// TIA Portal V15.1 program export: 6 tag tables, 0 data types, 10 data blocks, 37 code blocks (in call order from the OBs), 86 instance data blocks

VAR_GLOBAL   // PLC tag table "Analog"
   AI_AG AT %IW68 : Int;
   AI_FD AT %IW70 : Int;
   AI_AP AT %IW72 : Int;
   AI_SB AT %IW74 : Int;
   AI_TEMP_TL AT %IW76 : Int;
   AI_TEMP_AG AT %IW78 : Int;
   AI_TEMP_TS AT %IW80 : Int;
   AI_TEMP_AP AT %IW82 : Int;
   BT_SPAN_Riasing AT %M2.0 : Bool;
   BT_ZERO_Raising AT %M2.1 : Bool;
   MANUAL_Raissing AT %M2.2 : Bool;
   AI_IND_AGG1 AT %IW100 : Int;
   AI_IND_AGG2 AT %IW102 : Int;
   AI_IND_AGG3 AT %IW104 : Int;
   AI_IND_AGG4 AT %IW106 : Int;
   AI_IND_AGG5 AT %IW108 : Int;
END_VAR

VAR_GLOBAL   // PLC tag table "Default tag table"
END_VAR

VAR_GLOBAL   // PLC tag table "Default tag table_1"
   System_Byte AT %MB1 : Byte;
   FirstScan AT %M1.0 : Bool;
   DiagStatusUpdate AT %M1.1 : Bool;
   AlwaysTRUE AT %M1.2 : Bool;
   AlwaysFALSE AT %M1.3 : Bool;
   Clock_Byte AT %MB0 : Byte;
   Clock_10Hz AT %M0.0 : Bool;
   Clock_5Hz AT %M0.1 : Bool;
   "Clock_2.5Hz" AT %M0.2 : Bool;
   Clock_2Hz AT %M0.3 : Bool;
   "Clock_1.25Hz" AT %M0.4 : Bool;
   Clock_1Hz AT %M0.5 : Bool;
   "Clock_0.625Hz" AT %M0.6 : Bool;
   "Clock_0.5Hz" AT %M0.7 : Bool;
   "NAP LIEU" AT %M200.0 : Bool;
   "RUA NOI" AT %M200.1 : Bool;
   TH_NAP_WAG AT %M300.0 : Bool;
   TH_NAP_WAP AT %M300.2 : Bool;
   TH_NAP_WFD AT %M300.1 : Bool;
   TH_NAP_WSB AT %M300.3 : Bool;
   "LUU_CAN TAY" AT %M200.2 : Bool;
   "LUU TAY CEM1" AT %M200.3 : Bool;
   "LUU TAY CEM2" AT %M200.4 : Bool;
   "LUU TAY WAT1" AT %M200.5 : Bool;
   "LUU TAY ADD1" AT %M200.6 : Bool;
   XA_HET_AGG AT %M200.7 : Bool;
   "LUU TAY WAG1" AT %M210.0 : Bool;
   "LUU TAY WAG2" AT %M210.1 : Bool;
   "LUU TAY WAG3" AT %M210.2 : Bool;
   "LUU TAY WAG4" AT %M210.3 : Bool;
   "LUU TAY WAG5" AT %M210.4 : Bool;
END_VAR
VAR_GLOBAL CONSTANT   // user constants
   "Local(1)" : Hw_SubModule := 50;
   "Local~PROFINET_interface_1(1)" : Hw_Interface := 64;
   "Local~PROFINET_interface_1~Port_1(1)" : Hw_Interface := 65;
   "Local~HSC_1(1)" : Hw_Hsc := 257;
   "Local~HSC_2(1)" : Hw_Hsc := 258;
   "Local~HSC_3(1)" : Hw_Hsc := 259;
   "Local~HSC_4(1)" : Hw_Hsc := 260;
   "Local~HSC_5(1)" : Hw_Hsc := 261;
   "Local~HSC_6(1)" : Hw_Hsc := 262;
   "Local~AI_2_1(1)" : Hw_SubModule := 263;
   "Local~DI_14_DQ_10_1(1)" : Hw_SubModule := 264;
   "Local~Pulse_1(1)" : Hw_Pwm := 265;
   "Local~Pulse_2(1)" : Hw_Pwm := 266;
   "OB_Main_P1(1)" : OB_PCYCLE := 1;
   "Local~Pulse_3(1)" : Hw_Pwm := 267;
   "Local~Pulse_4(1)" : Hw_Pwm := 268;
   "None(1)" : Pip := 65535;
   "Automatic update(1)" : Pip := 0;
   "PIP 1(1)" : Pip := 1;
   "PIP 2(1)" : Pip := 2;
   "PIP 3(1)" : Pip := 3;
   "PIP 4(1)" : Pip := 4;
   "PIP OB Servo(1)" : Pip := 32768;
   "Local~DQ_8xRelay_1(1)" : Hw_SubModule := 273;
   "Local~AI_4x13BIT_1(1)" : Hw_SubModule := 271;
   "Local~AI_4xTC_1(1)" : Hw_SubModule := 272;
   "Local~DI_8_DQ_8x24VDC_1" : Hw_SubModule := 274;
   "Local~DQ_16xRelay_1(1)" : Hw_SubModule := 269;
   "Local~AI_4x13BIT_2(1)" : Hw_SubModule := 270;
END_VAR

VAR_GLOBAL   // PLC tag table "In_Put"
   "I_TH. NOI TRON" AT %I0.0 : Bool;   // Input_Tín hiệu nồi trộn
   "I_TH. BTX" AT %I0.1 : Bool;   // Input_Tín hiệu băng tải xiên
   "I_TH. BTN" AT %I0.2 : Bool;   // Input_Tín hiệu băng tải ngang
   "I_TH. TANG SAY" AT %I0.3 : Bool;   // Input_Tín hiệu tang sấy cốt liệu
   "I_TH. GAU COT LIEU" AT %I0.4 : Bool;   // Input_Tín hiệu gàu tải cốt liệu nóng
   "I_TH. GAU F/D" AT %I0.5 : Bool;   // Input_Tín hiệu gàu tải phụ gia bột
   "I_TH. SANG RUNG" AT %I0.6 : Bool;   // Input_Tín hiệu sàng rung cốt liệu nóng
   "I_TH. CUA DONG" AT %I0.7 : Bool;   // Input_Tín hiệu cửa nồi trộn đóng
   "I_TH. CUA MO" AT %I1.0 : Bool;   // Input_Tín hiệu cửa nồi trộn mở
   "I_TH. MNK" AT %I1.1 : Bool;   // Input_Tín hiệu máy nén khí chạy
   "I_TH. TRAN AG1" AT %I1.2 : Bool;   // Input_Tín hiệu báo tràn silo AG1
   "I_TH. TRAN AG2" AT %I1.3 : Bool;   // Input_Tín hiệu báo tràn silo AG2
   "I_TH. TRAN AG3" AT %I1.4 : Bool;   // Input_Tín hiệu báo tràn silo AG3
   "I_TH. TRAN AG4" AT %I1.5 : Bool;   // Input_Tín hiệu báo tràn silo AG4
   "I_TH. TRAN AG5" AT %I2.0 : Bool;   // Input_Tín hiệu báo tràn silo AG5
   "I_TH. TRAN FD1" AT %I2.1 : Bool;   // Input_Tín hiệu báo tràn silo F/D
   "I_TH. TRAN SB1" AT %I2.2 : Bool;   // Input_Tín hiệu báo tràn silo SBS
   "I_TH. SILO FD HIGHT" AT %I2.3 : Bool;   // Input_Tín hiệu báo mức cao silo chứa F/D
   "I_TH. SILO FD LOW" AT %I2.4 : Bool;   // Input_Tín hiệu báo mức thấp silo chứa F/D
   "TH. NOI TRON" AT %M400.0 : Bool;   // Tín hiệu nồi trộn
   "TH. BTX" AT %M400.1 : Bool;   // Tín hiệu băng tải xiên
   "TH. BTN" AT %M400.2 : Bool;   // Tín hiệu băng tải ngang
   "TH. TANG SAY" AT %M400.3 : Bool;   // Tín hiệu tang sấy cốt liệu
   "TH. GAU COT LIEU" AT %M400.4 : Bool;   // Tín hiệu gàu tải cốt liệu nóng
   "TH. GAU F/D" AT %M400.5 : Bool;   // Tín hiệu gàu tải phụ gia bột
   "TH. SANG RUNG" AT %M400.6 : Bool;   // Tín hiệu sàng rung cốt liệu nóng
   "TH. CUA DONG" AT %M400.7 : Bool;   // Tín hiệu cửa nồi trộn đóng
   "TH. CUA MO" AT %M401.0 : Bool;   // Tín hiệu cửa nồi trộn mở
   "TH. MNK" AT %M401.1 : Bool;   // Tín hiệu máy nén khí chạy
   "TH. TRAN AG1" AT %M401.2 : Bool;   // Tín hiệu báo tràn silo AG1
   "TH. TRAN AG2" AT %M401.3 : Bool;   // Tín hiệu báo tràn silo AG2
   "TH. TRAN AG3" AT %M401.4 : Bool;   // Tín hiệu báo tràn silo AG3
   "TH. TRAN AG4" AT %M401.5 : Bool;   // Tín hiệu báo tràn silo AG4
   "TH. TRAN AG5" AT %M401.6 : Bool;   // Tín hiệu báo tràn silo AG5
   "TH. TRAN FD1" AT %M401.7 : Bool;   // Tín hiệu báo tràn silo F/D
   "TH. TRAN SB1" AT %M402.0 : Bool;   // Tín hiệu báo tràn silo SBS
   "TH. SILO FD HIGHT" AT %M402.1 : Bool;   // Tín hiệu báo mức cao silo chứa F/D
   "TH. SILO FD LOW" AT %M402.2 : Bool;   // Tín hiệu báo mức thấp silo chứa F/D
   "TH_CNM SIM" AT %M402.3 : Bool;
   "TH_CND SIM" AT %M402.4 : Bool;
END_VAR

VAR_GLOBAL   // PLC tag table "Out_Put"
   "Q_CAN AP1" AT %Q4.0 : Bool;   // Output_Nồi trộn
   "Q_GAU COT LIEU" AT %Q0.5 : Bool;   // Output_Băng tải xiên
   Q_BTX AT %Q0.1 : Bool;   // Output_Băng tải ngang
   Q_BTN AT %Q0.2 : Bool;   // Output_Tang sấy cốt liệu
   "Q_TANG SAY" AT %Q0.3 : Bool;   // Output_Bơm dầu DO
   "Q_XA W_AG1" AT %Q4.2 : Bool;   // Output_Gàu tải cốt liệu nóng
   "Q_XA W_SB1" AT %Q4.5 : Bool;   // Output_Sàn rung cốt liệu
   "Q_BOM NUOC" AT %Q2.1 : Bool;   // Output_Gàu tải phụ F/D
   "Q_MO CUA" AT %Q2.2 : Bool;   // Output_Vít tải F/D
   "Q_XA CL5" AT %Q3.1 : Bool;   // Output_Bơm nạp hạt nhựa SBS
   "Q_DONG CUA" AT %Q2.3 : Bool;   // Output_Quạt gió lọc bụi
   Q_MNK AT %Q2.4 : Bool;   // Output_Bơm nước lọc bụi
   "Q_BOM SBS" AT %Q1.1 : Bool;   // Output_Van mở cửa nồi trộn
   "Q_CAN AG1" AT %Q3.2 : Bool;   // Output_Van đóng cửa nồi trộn
   "Q_VIT TAI FD" AT %Q1.0 : Bool;   // Output_Máy nén khí
   "Q_XA CL1" AT %Q2.5 : Bool;   // Output_Băng tải xả cốt liệu 1
   "Q_XA CL2" AT %Q2.6 : Bool;   // Output_Băng tải xả cốt liệu 2
   "Q_CAN AG2" AT %Q3.3 : Bool;   // Output_Băng tải xả cốt liệu 3
   "Q_XA CL3" AT %Q2.7 : Bool;   // Output_Băng tải xả cốt liệu 4
   "Q_XA CL4" AT %Q3.0 : Bool;   // Output_Băng tải xả cốt liệu 5
   "Q_CAN AG3" AT %Q3.4 : Bool;   // Output_Van cân AG1
   "Q_CAN AG4" AT %Q3.5 : Bool;   // Output_Van cân AG2
   "Q_CAN AG5" AT %Q3.6 : Bool;   // Output_Van cân AG3
   "Q_SAN RUNG" AT %Q0.6 : Bool;   // Output_Van cân AG4
   "Q_CAN FD1" AT %Q3.7 : Bool;   // Output_Van cân AG5
   "Q_CAN SB1" AT %Q4.1 : Bool;   // Output_Van cân F/D
   "Q_NOI TRON" AT %Q0.0 : Bool;   // Output_Bơm nhựa
   "Q_XA W_AP1" AT %Q4.4 : Bool;   // Output_Van cân hạt nhựa SBS
   "Q_XA W_FD1" AT %Q4.3 : Bool;   // Output_Van xả cân AG1
   "Q_BOM TUOI NHUA" AT %Q4.6 : Bool;   // Output_Van xả cân FD1
   "Q_DAU DOT" AT %Q4.7 : Bool;   // Output_Van xả cân AP1
   "Q_VAN XA SBS" AT %Q5.0 : Bool;   // Output_Van xả cân SB1
   "Q_Rung CL1" AT %Q5.1 : Bool;   // Output_Bổ ssung 1
   "Q_Rung CL2" AT %Q5.2 : Bool;   // Output_Bổ ssung 2
   "Q_Rung CL3" AT %Q5.3 : Bool;   // Output_Bổ ssung 3
   "Q_NOTE 7" AT %Q5.4 : Bool;   // Output_Bổ ssung 4
   "Q_QUAT GIO" AT %Q2.0 : Bool;   // Output_Bổ ssung 5
   "Q_GAU FD" AT %Q0.7 : Bool;   // Output_Bổ ssung 6
   "Q_BOM DAU" AT %Q0.4 : Bool;   // Output_Bổ ssung 7
   "NOI TRON" AT %M500.0 : Bool;   // Nồi trộn
   BTX AT %M500.1 : Bool;   // Băng tải xiên
   BTN AT %M500.2 : Bool;   // Băng tải ngang
   "TANG SAY" AT %M500.3 : Bool;   // Tang sấy cốt liệu
   "BOM DAU" AT %M500.4 : Bool;   // Bơm dầu DO
   "GAU COT LIEU" AT %M500.5 : Bool;   // Gàu tải cốt liệu nóng
   "SAN RUNG" AT %M500.6 : Bool;   // Sàn rung cốt liệu
   "GAU FD" AT %M500.7 : Bool;   // Gàu tải phụ F/D
   "VIT TAI FD" AT %M501.0 : Bool;   // Vít tải F/D
   "BOM SBS" AT %M501.1 : Bool;   // Bơm nạp hạt nhựa SBS
   "QUAT GIO" AT %M501.2 : Bool;   // Quạt gió lọc bụi
   "BOM NUOC" AT %M501.3 : Bool;   // Bơm nước lọc bụi
   "MO CUA" AT %M501.4 : Bool;   // Van mở cửa nồi trộn
   "DONG CUA" AT %M501.5 : Bool;   // Van đóng cửa nồi trộn
   MNK AT %M501.6 : Bool;   // Máy nén khí
   "XA CL1" AT %M501.7 : Bool;   // Băng tải xả cốt liệu 1
   "XA CL2" AT %M502.0 : Bool;   // Băng tải xả cốt liệu 2
   "XA CL3" AT %M502.1 : Bool;   // Băng tải xả cốt liệu 3
   "XA CL4" AT %M502.2 : Bool;   // Băng tải xả cốt liệu 4
   "XA CL5" AT %M502.3 : Bool;   // Băng tải xả cốt liệu 5
   "CAN AG1" AT %M502.4 : Bool;   // Van cân AG1
   "CAN AG2" AT %M502.5 : Bool;   // Van cân AG2
   "CAN AG3" AT %M502.6 : Bool;   // Van cân AG3
   "CAN AG4" AT %M502.7 : Bool;   // Van cân AG4
   "CAN AG5" AT %M503.0 : Bool;   // Van cân AG5
   "CAN FD1" AT %M503.1 : Bool;   // Van cân F/D
   "CAN AP1" AT %M503.2 : Bool;   // Bơm nhựa
   "CAN SB1" AT %M503.3 : Bool;   // Van cân hạt nhựa SBS
   "XA W_AG1" AT %M503.4 : Bool;   // Van xả cân AG1
   "XA W_FD1" AT %M503.5 : Bool;   // Van xả cân FD1
   "XA W_AP1" AT %M503.6 : Bool;   // Van xả cân AP1
   "XA W_SB1" AT %M503.7 : Bool;   // Van xả cân SB1
   "BOM TUOI NHUA" AT %M504.0 : Bool;   // Bổ ssung 1
   "DAU DOT" AT %M504.1 : Bool;   // Bổ ssung 2
   "VAN XA SBS" AT %M504.2 : Bool;   // Bổ ssung 3
   "RUNG CL1" AT %M504.3 : Bool;   // Bổ ssung 4
   "RUNG CL2" AT %M504.4 : Bool;   // Bổ ssung 5
   "RUNG CL3" AT %M504.5 : Bool;   // Bổ ssung 6
   "NOTE 7" AT %M504.6 : Bool;   // Bổ ssung 7
   "Q_XA W_IND AGG1" AT %Q6.0 : Bool;   // Mode=độc lập, Van xả cấn AGG1
   "Q_XA W_IND AGG2" AT %Q6.1 : Bool;   // Mode=độc lập, Van xả cấn AGG2
   "Q_XA W_IND AGG3" AT %Q6.2 : Bool;   // Mode=độc lập, Van xả cấn AGG3
   "Q_XA W_IND AGG4" AT %Q6.3 : Bool;   // Mode=độc lập, Van xả cấn AGG4
   "Q_XA W_IND AGG5" AT %Q6.4 : Bool;   // Mode=độc lập, Van xả cấn AGG5
END_VAR

VAR_GLOBAL   // PLC tag table "XUNG_TEMP"
   P_AGG1_EM AT %M100.0 : Bool;
   P_AGG2_EM AT %M100.1 : Bool;
   P_AGG3_EM AT %M100.2 : Bool;
   P_AGG4_EM AT %M100.3 : Bool;
   P_AGG5_EM AT %M100.4 : Bool;
   P_AGG6_EM AT %M100.5 : Bool;
   P_CE1_EM AT %M100.6 : Bool;
   P_CE2_EM AT %M100.7 : Bool;
   P_CE3_EM AT %M101.0 : Bool;
   P_CE4_EM AT %M101.1 : Bool;
   P_CE5_EM AT %M101.2 : Bool;
   P_WA1_EM AT %M101.3 : Bool;
   P_WA2_EM AT %M101.4 : Bool;
   P_ADD1_EM AT %M101.5 : Bool;
   P_ADD2_EM AT %M101.6 : Bool;
   P_ADD3_EM AT %M101.7 : Bool;
   P_ADD4_EM AT %M102.0 : Bool;
   P_ADD5_EM AT %M102.1 : Bool;
   P_ADD6_EM AT %M102.2 : Bool;
   P_WAGG1_EM AT %M102.3 : Bool;
   P_WAGG2_EM AT %M102.4 : Bool;
   P_WAGG3_EM AT %M102.5 : Bool;
   P_WAGG4_EM AT %M102.6 : Bool;
   P_WAGG5_EM AT %M102.7 : Bool;
   P_WAGG6_EM AT %M103.0 : Bool;
   P_WCEM1_EM AT %M103.1 : Bool;
   P_WCEM2_EM AT %M103.2 : Bool;
   P_WWAT1_EM AT %M103.3 : Bool;
   P_WWAT2_EM AT %M103.4 : Bool;
   P_WADD1_EM AT %M103.5 : Bool;
   P_WADD2_EM AT %M103.6 : Bool;
   P_AGG1_FU AT %M103.7 : Bool;
   P_AGG2_FU AT %M104.0 : Bool;
   P_AGG3_FU AT %M104.1 : Bool;
   P_AGG4_FU AT %M104.2 : Bool;
   P_AGG5_FU AT %M104.3 : Bool;
   P_AGG6_FU AT %M104.4 : Bool;
   P_CE1_FU AT %M104.5 : Bool;
   P_CE2_FU AT %M104.6 : Bool;
   P_CE3_FU AT %M104.7 : Bool;
   P_CE4_FU AT %M105.0 : Bool;
   P_CE5_FU AT %M105.1 : Bool;
   P_WA1_FU AT %M105.2 : Bool;
   P_WA2_FU AT %M105.3 : Bool;
   P_ADD1_FU AT %M105.4 : Bool;
   P_ADD2_FU AT %M105.5 : Bool;
   P_ADD3_FU AT %M105.6 : Bool;
   P_ADD4_FU AT %M105.7 : Bool;
   P_ADD5_FU AT %M106.0 : Bool;
   P_ADD6_FU AT %M106.1 : Bool;
   P_WAGG1_FU AT %M106.2 : Bool;
   P_WAGG2_FU AT %M106.3 : Bool;
   P_WAGG3_FU AT %M106.4 : Bool;
   P_WAGG4_FU AT %M106.5 : Bool;
   P_WAGG5_FU AT %M106.6 : Bool;
   P_WAGG6_FU AT %M106.7 : Bool;
   P_WCEM1_FU AT %M107.0 : Bool;
   P_WCEM2_FU AT %M107.1 : Bool;
   P_WWAT1_FU AT %M107.2 : Bool;
   P_WWAT2_FU AT %M107.3 : Bool;
   P_WADD1_FU AT %M107.4 : Bool;
   P_WADD2_FU AT %M107.5 : Bool;
   P_PTG_EM AT %M107.6 : Bool;
   P_PTG_FU AT %M107.7 : Bool;
   P_SKIP_EM AT %M108.0 : Bool;
   P_SKIP_FU AT %M108.1 : Bool;
   P_MIXER_EM AT %M108.2 : Bool;
   P_MIXER_FU AT %M108.3 : Bool;
   P_RUN AT %M108.4 : Bool;
   "P_COT LIEU_FU" AT %M108.5 : Bool;
   "P_COT LIEU_EM" AT %M108.6 : Bool;
   "P_XA AGG1" AT %M108.7 : Bool;
   "P_XA AGG2" AT %M109.0 : Bool;
   "P_XA AGG3" AT %M109.1 : Bool;
   "P_XA AGG4" AT %M109.2 : Bool;
   "P_XA AGG5" AT %M109.3 : Bool;
   "P_XA AGG6" AT %M109.4 : Bool;
   "P_XA PTG" AT %M109.5 : Bool;
   "P_XA CEM1" AT %M109.6 : Bool;
   "P_XA CEM2" AT %M109.7 : Bool;
   "P_XA WAT1" AT %M110.0 : Bool;
   "P_XA WAT2" AT %M110.1 : Bool;
   "P_XA ADD1" AT %M110.2 : Bool;
   "P_XA ADD2" AT %M110.3 : Bool;
END_VAR

DATA_BLOCK "C#1_RB"   // DB1
{ S7_Optimized_Access := 'FALSE' }
VERSION : 0.1
// stored: AutoNumber true, CodeModifiedDate 2024-10-21T16:21:19.3207346Z, CompileDate 2025-08-30T17:40:33.1183285Z, CreationDate 2024-10-12T12:36:08.0193576Z, DBAccessibleFromOPCUA true, InterfaceModifiedDate 2024-10-21T16:21:19.3207346Z, IsConsistent true, IsKnowHowProtected false, IsOnlyStoredInLoadMemory false, IsPLCDB false, IsWriteProtectedInAS false, ModifiedDate 2024-10-21T16:21:19.3207346Z, ParameterModified 2024-10-21T16:21:19.3207346Z, StructureModified 2024-10-21T16:21:19.3207346Z
   VAR
      "TH. NOI TRON" : Bool;   // Tín hiệu nồi trộn
      "TH. BTX" : Bool;   // Tín hiệu băng tải xiên
      "TH. BTN" : Bool;   // Tín hiệu băng tải ngang
      "TH. TANG SAY" : Bool;   // Tín hiệu tang sấy cốt liệu
      "TH. GAU COT LIEU" : Bool;   // Tín hiệu gàu tải cốt liệu nóng
      "TH. GAU F/D" : Bool;   // Tín hiệu gàu tải phụ gia bột
      "TH. SAN RUNG" : Bool;   // Tín hiệu sàng rung cốt liệu nóng
      "TH. CUA DONG" : Bool;   // Tín hiệu cửa nồi trộn đóng
      "TH. CUA MO" : Bool;   // Tín hiệu cửa nồi trộn mở
      "TH. MNK" : Bool;   // Tín hiệu máy nén khí chạy
      "TH. TRAN AG1" : Bool;   // Tín hiệu báo tràn silo AG1
      "TH. TRAN AG2" : Bool;   // Tín hiệu báo tràn silo AG2
      "TH. TRAN AG3" : Bool;   // Tín hiệu báo tràn silo AG3
      "TH. TRAN AG4" : Bool;   // Tín hiệu báo tràn silo AG4
      "TH. TRAN AG5" : Bool;   // Tín hiệu báo tràn silo AG5
      "TH. TRAN FD1" : Bool;   // Tín hiệu báo tràn silo F/D
      "TH. TRAN SB1" : Bool;   // Tín hiệu báo tràn silo SBS
      "TH. SILO FD HIGHT" : Bool;   // Tín hiệu báo mức cao silo chứa F/D
      "TH. SILO FD LOW" : Bool;   // Tín hiệu báo mức thấp silo chứa F/D
      "NOI TRON" : Bool;   // Nồi trộn
      BTX : Bool;   // Băng tải xiên
      BTN : Bool;   // Băng tải ngang
      "TANG SAY" : Bool;   // Tang sấy cốt liệu
      "BOM DAU" : Bool;   // Bơm dầu DO
      "GAU COT LIEU" : Bool;   // Gàu tải cốt liệu nóng
      "SAN RUNG" : Bool;   // Sàn rung cốt liệu
      "GAU FD" : Bool;   // Gàu tải phụ F/D
      "VIT TAI FD" : Bool;   // Vít tải F/D
      "BOM SBS" : Bool;   // Bơm nạp hạt nhựa SBS
      "QUAT GIO" : Bool;   // Quạt gió lọc bụi
      "BOM NUOC" : Bool;   // Bơm nước lọc bụi
      "MO CUA" : Bool;   // Van mở cửa nồi trộn
      "DONG CUA" : Bool;   // Van đóng cửa nồi trộn
      MNK : Bool;   // Máy nén khí
      "XA CL1" : Bool;   // Băng tải xả cốt liệu 1
      "XA CL2" : Bool;   // Băng tải xả cốt liệu 2
      "XA CL3" : Bool;   // Băng tải xả cốt liệu 3
      "XA CL4" : Bool;   // Băng tải xả cốt liệu 4
      "XA CL5" : Bool;   // Băng tải xả cốt liệu 5
      "CAN AG1" : Bool;   // Van cân AG1
      "CAN AG2" : Bool;   // Van cân AG2
      "CAN AG3" : Bool;   // Van cân AG3
      "CAN AG4" : Bool;   // Van cân AG4
      "CAN AG5" : Bool;   // Van cân AG5
      "CAN FD1" : Bool;   // Van cân F/D
      "CAN AP1" : Bool;   // Bơm nhựa
      "CAN SB1" : Bool;   // Van cân hạt nhựa SBS
      "XA W_AG1" : Bool;   // Van xả cân AG1
      "XA W_FD1" : Bool;   // Van xả cân FD1
      "XA W_AP1" : Bool;   // Van xả cân AP1
      "XA W_SB1" : Bool;   // Van xả cân SB1
      BOM_TUOI_NHUA : Bool;   // Bổ sung 1
      DAU_DOT : Bool;   // Bổ sung 2
      VAN_PNSBS : Bool;   // Bổ sung 3
      "RUNG CL1" : Bool;   // Bổ sung 4
      "RUNG CL2" : Bool;   // Bổ sung 5
      "RUNG CL3" : Bool;   // Bổ sung 6
      "NOTE 7" : Bool;   // Bổ sung 7
      RUNNING : Bool;   // Trạng thái đang trộn
      SIMULATION : Bool;   // Trạng thái chạy mô phỏng
      MIXER_FULL : Bool;   // Trạng thái nồi trộn báo đầy
      TTC_AG1 : Bool;   // Trạng thái cân Ag1
      TTC_AG2 : Bool;   // Trạng thái cân Ag2
      TTC_AG3 : Bool;   // Trạng thái cân Ag3
      TTC_AG4 : Bool;   // Trạng thái cân Ag4
      TTC_AG5 : Bool;   // Trạng thái cân Ag5
      TTC_FD1 : Bool;   // Trạng thái cân FD1
      TTC_AP1 : Bool;   // Trạng thái cân AP1
      TTC_SB1 : Bool;   // Trạng thái cân SBS1
   END_VAR
BEGIN
END_DATA_BLOCK

DATA_BLOCK "C#2_WB"   // DB2
{ S7_Optimized_Access := 'FALSE' }
VERSION : 0.1
// stored: AutoNumber true, CodeModifiedDate 2026-01-04T14:05:19.1281212Z, CompileDate 2026-01-04T14:27:04.768919Z, CreationDate 2024-10-12T12:36:08.0193576Z, DBAccessibleFromOPCUA true, InterfaceModifiedDate 2026-01-04T14:05:19.1281212Z, IsConsistent true, IsKnowHowProtected false, IsOnlyStoredInLoadMemory false, IsPLCDB false, IsWriteProtectedInAS false, ModifiedDate 2026-01-04T14:05:19.1281212Z, ParameterModified 2026-01-04T14:05:19.1281212Z, StructureModified 2026-01-04T14:05:19.1281212Z
   VAR
      F1_NN_RUN : Bool;   // F1 Nút nhấn chạy
      F2_SW_PAU : Bool;   // F2 Công tắc tạm dừng
      F3_NN_STOP : Bool;   // F3 Nút nhấn dừng/hủy mẻ
      F4_SW_SIM : Bool;   // F4 Công tắc chế độ mô phỏng
      "SW_MAN/AUTO" : Bool;   // Công tắc chế độ chạy tay/tự động
      SW_XA_LIEU : Bool;   // Công tắc chế độ xả cân cốt liệu
      SW_NAP_NOI_TRON : Bool;   // Công tắc nạp liệu nồi trộn
      SW_XA_NOI_TRON : Bool;   // Công tắc chế độ xả bê tông
      "NN_NOI TRON" : Bool;   // Nút nhấn Nồi trộn
      NN_BTX : Bool;   // Nút nhấn Băng tải xiên
      NN_BTN : Bool;   // Nút nhấn Băng tải ngang
      "NN_TANG SAY" : Bool;   // Nút nhấn Tang sấy cốt liệu
      "NN_BOM DAU" : Bool;   // Nút nhấn Bơm dầu DO
      "NN_GAU COT LIEU" : Bool;   // Nút nhấn Gàu tải cốt liệu nóng
      "NN_SAN RUNG" : Bool;   // Nút nhấn Sàn rung cốt liệu
      "NN_GAU FD" : Bool;   // Nút nhấn Gàu tải phụ F/D
      "NN_VIT TAI FD" : Bool;   // Nút nhấn Vít tải F/D
      "NN_BOM SBS" : Bool;   // Nút nhấn Bơm nạp hạt nhựa SBS
      "NN_QUAT GIO" : Bool;   // Nút nhấn Quạt gió lọc bụi
      "NN_BOM NUOC" : Bool;   // Nút nhấn Bơm nước lọc bụi
      "NN_MO CUA" : Bool;   // Nút nhấn Van mở cửa nồi trộn
      "NN_DONG CUA" : Bool;   // Nút nhấn Van đóng cửa nồi trộn
      NN_MNK : Bool;   // Nút nhấn Máy nén khí
      "SW_XA CL1" : Bool;   // Công tắc Băng tải xả cốt liệu 1
      "SW_XA CL2" : Bool;   // Công tắc Băng tải xả cốt liệu 2
      "SW_XA CL3" : Bool;   // Công tắc Băng tải xả cốt liệu 3
      "SW_XA CL4" : Bool;   // Công tắc Băng tải xả cốt liệu 4
      "SW_XA CL5" : Bool;   // Công tắc Băng tải xả cốt liệu 5
      "NN_CAN AG1" : Bool;   // Nút nhấn Van cân AG1
      "NN_CAN AG2" : Bool;   // Nút nhấn Van cân AG2
      "NN_CAN AG3" : Bool;   // Nút nhấn Van cân AG3
      "NN_CAN AG4" : Bool;   // Nút nhấn Van cân AG4
      "NN_CAN AG5" : Bool;   // Nút nhấn Van cân AG5
      "NN_CAN FD1" : Bool;   // Nút nhấn Van cân F/D
      "NN_CAN AP1" : Bool;   // Nút nhấn Bơm nhựa
      "NN_CAN SB1" : Bool;   // Nút nhấn Van cân hạt nhựa SBS
      "SW_XA W_AG1" : Bool;   // Công tắc Van xả cân AG1
      "SW_XA W_FD1" : Bool;   // Công tắc Van xả cân FD1
      "SW_XA W_AP1" : Bool;   // Công tắc Van xả cân AP1
      "SW_XA W_SB1" : Bool;   // Công tắc Van xả cân SB1
      "NN_BOM TUOI NHUA" : Bool;   // Nút nhấn Bổ sung 1
      "NN_XA HET AGG" : Bool;   // Nút nhấn Bổ sung 2
      "NN_DAU DOT" : Bool;   // Nút nhấn Bổ sung 3
      NN_VAN_PNSBS : Bool;   // Nút nhấn Bổ sung 4
      "NN_NOTE 5" : Bool;   // Nút nhấn Bổ sung 5
      "NN_NOTE 6" : Bool;   // Nút nhấn Bổ sung 6
      "NN_NOTE 7" : Bool;   // Nút nhấn Bổ sung 7
      NN_FU_AG1 : Bool;   // Nút nhấn Báo đầy silo AG1
      NN_FU_AG2 : Bool;   // Nút nhấn Báo đầy silo AG2
      NN_FU_AG3 : Bool;   // Nút nhấn Báo đầy silo AG3
      NN_FU_AG4 : Bool;   // Nút nhấn Báo đầy silo AG4
      NN_FU_AG5 : Bool;   // Nút nhấn Báo đầy silo AG5
      NN_FU_FD1 : Bool;   // Nút nhấn Báo đầy silo FD1
      NN_FU_AP1 : Bool;   // Nút nhấn Báo đầy silo AP1
      NN_FU_SB1 : Bool;   // Nút nhấn Báo đầy silo SBS1
      SW_PA_AG1 : Bool;   // Công tắc Tạm dừng cân AG1
      SW_PA_AG2 : Bool;   // Công tắc Tạm dừng cân AG2
      SW_PA_AG3 : Bool;   // Công tắc Tạm dừng cân AG3
      SW_PA_AG4 : Bool;   // Công tắc Tạm dừng cân AG4
      SW_PA_AG5 : Bool;   // Công tắc Tạm dừng cân AG5
      SW_PA_FD1 : Bool;   // Công tắc Tạm dừng cân FD1
      SW_PA_AP1 : Bool;   // Công tắc Tạm dừng cân AP1
      SW_PA_SB1 : Bool;   // Công tắc Tạm dừng cân SBS1
      NN_ZERO_AG1 : Bool;   // Nút nhấn chỉnh 0 cân AG1
      NN_SPAN_AG1 : Bool;   // Nút nhấn chỉnh tải cân AG1
      NN_ZERO_FD1 : Bool;   // Nút nhấn chỉnh 0 cân FD1
      NN_SPAN_FD1 : Bool;   // Nút nhấn chỉnh tải cân FD1
      NN_ZERO_AP1 : Bool;   // Nút nhấn chỉnh 0 cân AP1
      NN_SPAN_AP1 : Bool;   // Nút nhấn chỉnh tải cân AP1
      NN_ZERO_SB1 : Bool;   // Nút nhấn chỉnh 0 cân SBS1
      NN_SPAN_SB1 : Bool;   // Nút nhấn chỉnh tải cân SBS1
      "NN_ZERO_TEMP TS" : Bool;   // Nút nhấn chỉnh 0 nhiệt độ 1
      "NN_SPAN_TEMP TS" : Bool;   // Nút nhấn chỉnh tải nhiệt độ 1
      "NN_ZERO_TEMP AG" : Bool;   // Nút nhấn chỉnh 0 nhiệt độ 2
      "NN_SPAN_TEMP AG" : Bool;   // Nút nhấn chỉnh tải nhiệt độ 2
      "NN_ZERO_TEMP AP" : Bool;   // Nút nhấn chỉnh 0 nhiệt độ 3
      "NN_SPAN_TEMP AP" : Bool;   // Nút nhấn chỉnh tải nhiệt độ 3
      "NN_ZERO_TEMP TL" : Bool;   // Nút nhấn chỉnh 0 nhiệt độ 4
      "NN_SPAN_TEMP TL" : Bool;   // Nút nhấn chỉnh tải nhiệt độ 4
      "NN_RUNG AG1" : Bool;   // Nút nhấn rung phễu cân AG1
      "NN_RUNG FD1" : Bool;   // Nút nhấn rung phễu cân FD1
      "NN_RUNG SB1" : Bool;   // Nút nhấn rung phễu cân SBS1
      "XAC NHAN CAN DU" : Bool;   // Nút nhấn xác nhận cân dư
      XNC_AUT_AG1 : Bool;   // Tự dộng xác nhận cân dư Agg1
      XNC_AUT_AG2 : Bool;   // Tự dộng xác nhận cân dư Agg2
      XNC_AUT_AG3 : Bool;   // Tự dộng xác nhận cân dư Agg3
      XNC_AUT_AG4 : Bool;   // Tự dộng xác nhận cân dư Agg4
      XNC_AUT_AG5 : Bool;   // Tự dộng xác nhận cân dư Agg5
      XNC_AUT_FD1 : Bool;   // Tự dộng xác nhận cân dư FD1
      XNC_AUT_AP1 : Bool;   // Tự dộng xác nhận cân dư AP1
      XNC_AUT_SB1 : Bool;   // Tự dộng xác nhận cân dư SBS1
      BUTRU_AGG1 : Bool;   // Bù trừ khối lượng Agg1
      BUTRU_AGG2 : Bool;   // Bù trừ khối lượng Agg2
      BUTRU_AGG3 : Bool;   // Bù trừ khối lượng Agg3
      BUTRU_AGG4 : Bool;   // Bù trừ khối lượng Agg4
      BUTRU_AGG5 : Bool;   // Bù trừ khối lượng Agg5
      BUTRU_FD1 : Bool;   // Bù trừ khối lượng FD1
      BUTRU_AP1 : Bool;   // Bù trừ khối lượng AP1
      BUTRU_SB1 : Bool;   // Bù trừ khối lượng SBS1
      "NN_RUNG CL1" : Bool;
      "NN_RUNG CL2" : Bool;
      "NN_RUNG CL3" : Bool;
      SETUP_MODE_DOC_LAP : Bool;   // OFF=cộng dồn, ON=độc lập
      NN_ZERO_IND_AG1 : Bool;
      NN_SPAN_IND_AG1 : Bool;
      NN_ZERO_IND_AG2 : Bool;
      NN_SPAN_IND_AG2 : Bool;
      NN_ZERO_IND_AG3 : Bool;
      NN_SPAN_IND_AG3 : Bool;
      NN_ZERO_IND_AG4 : Bool;
      NN_SPAN_IND_AG4 : Bool;
      NN_ZERO_IND_AG5 : Bool;
      NN_SPAN_IND_AG5 : Bool;
   END_VAR
BEGIN
END_DATA_BLOCK

DATA_BLOCK "C#3_WD_SILO"   // DB3
{ S7_Optimized_Access := 'FALSE' }
VERSION : 0.1
// stored: AutoNumber true, CodeModifiedDate 2024-09-25T15:44:48.8692886Z, CompileDate 2025-08-30T17:40:31.5137835Z, CreationDate 2024-10-12T12:36:08.0193576Z, DBAccessibleFromOPCUA true, InterfaceModifiedDate 2024-09-25T15:44:48.8692886Z, IsConsistent true, IsKnowHowProtected false, IsOnlyStoredInLoadMemory false, IsPLCDB false, IsWriteProtectedInAS false, ModifiedDate 2024-09-25T15:47:56.1309792Z, ParameterModified 2024-09-25T15:44:48.8692886Z, StructureModified 2024-09-25T15:44:48.8692886Z
   VAR RETAIN
      AG1_SS_TREN : Real;   // Ag1 sai số trên
      AG1_SS_DUOI : Real;   // Ag1 sai số dưới
      AG1_KL_RTD : Real;   // Ag1 khối lượng rơi tự do
      AG1_TG_ON_CAN : Real;   // Ag1 thời gian mở cân
      AG1_TG_OFF_CAN : Real;   // Ag1 thời gian đóng cân
      AG1_TG_ODC : Real;   // Ag1 thời gian tính lượng rơi thêm
      AG2_SS_TREN : Real;   // Ag2 sai số trên
      AG2_SS_DUOI : Real;   // Ag2 sai số dưới
      AG2_KL_RTD : Real;   // Ag2 khối lượng rơi tự do
      AG2_TG_ON_CAN : Real;   // Ag2 thời gian mở cân
      AG2_TG_OFF_CAN : Real;   // Ag2 thời gian đóng cân
      AG2_TG_ODC : Real;   // Ag2 thời gian tính lượng rơi thêm
      AG3_SS_TREN : Real;   // Ag3 sai số trên
      AG3_SS_DUOI : Real;   // Ag3 sai số dưới
      AG3_KL_RTD : Real;   // Ag3 khối lượng rơi tự do
      AG3_TG_ON_CAN : Real;   // Ag3 thời gian mở cân
      AG3_TG_OFF_CAN : Real;   // Ag3 thời gian đóng cân
      AG3_TG_ODC : Real;   // Ag3 thời gian tính lượng rơi thêm
      AG4_SS_TREN : Real;   // Ag4 sai số trên
      AG4_SS_DUOI : Real;   // Ag4 sai số dưới
      AG4_KL_RTD : Real;   // Ag4 khối lượng rơi tự do
      AG4_TG_ON_CAN : Real;   // Ag4 thời gian mở cân
      AG4_TG_OFF_CAN : Real;   // Ag4 thời gian đóng cân
      AG4_TG_ODC : Real;   // Ag4 thời gian tính lượng rơi thêm
      AG5_SS_TREN : Real;   // Ag5 sai số trên
      AG5_SS_DUOI : Real;   // Ag5 sai số dưới
      AG5_KL_RTD : Real;   // Ag5 khối lượng rơi tự do
      AG5_TG_ON_CAN : Real;   // Ag5 thời gian mở cân
      AG5_TG_OFF_CAN : Real;   // Ag5 thời gian đóng cân
      AG5_TG_ODC : Real;   // Ag5 thời gian tính lượng rơi thêm
      FD1_SS_TREN : Real;   // FD1 sai số trên
      FD1_SS_DUOI : Real;   // FD1 sai số dưới
      FD1_KL_RTD : Real;   // FD1 khối lượng rơi tự do
      FD1_TG_ON_CAN : Real;   // FD1 thời gian mở cân
      FD1_TG_OFF_CAN : Real;   // FD1 thời gian đóng cân
      FD1_TG_ODC : Real;   // FD1 thời gian tính lượng rơi thêm
      AP1_SS_TREN : Real;   // AP1 sai số trên
      AP1_SS_DUOI : Real;   // AP1 sai số dưới
      AP1_KL_RTD : Real;   // AP1 khối lượng rơi tự do
      AP1_TG_ON_CAN : Real;   // AP1 thời gian mở cân
      AP1_TG_OFF_CAN : Real;   // AP1 thời gian đóng cân
      AP1_TG_ODC : Real;   // AP1 thời gian tính lượng rơi thêm
      SB1_SS_TREN : Real;   // SBS1 sai số trên
      SB1_SS_DUOI : Real;   // SBS1 sai số dưới
      SB1_KL_RTD : Real;   // SBS1 khối lượng rơi tự do
      SB1_TG_ON_CAN : Real;   // SBS1 thời gian mở cân
      SB1_TG_OFF_CAN : Real;   // SBS1 thời gian đóng cân
      SB1_TG_ODC : Real;   // SBS1 thời gian tính lượng rơi thêm
   END_VAR
BEGIN
END_DATA_BLOCK

DATA_BLOCK "C#4_WD_WEIGHT"   // DB4
{ S7_Optimized_Access := 'FALSE' }
VERSION : 0.1
// stored: AutoNumber true, CodeModifiedDate 2024-09-25T16:02:28.9173662Z, CompileDate 2025-08-30T17:40:33.07032Z, CreationDate 2024-10-12T12:36:08.0193576Z, DBAccessibleFromOPCUA true, InterfaceModifiedDate 2024-09-25T16:02:28.9173662Z, IsConsistent true, IsKnowHowProtected false, IsOnlyStoredInLoadMemory false, IsPLCDB false, IsWriteProtectedInAS false, ModifiedDate 2024-10-13T07:08:48.1421634Z, ParameterModified 2024-09-25T16:02:28.9173662Z, StructureModified 2024-09-25T16:02:28.9173662Z
   VAR RETAIN
      "W_AG1_TG.DLC" : Real;   // Phễu cân Cốt liệu 1_Thời gian trễ cân
      "W_AG1_TG.DLX" : Real;   // Phễu cân Cốt liệu 1_Thời gian trễ xả
      "W_AG1_TG.DLD" : Real;   // Phễu cân Cốt liệu 1_Thời gian trễ đóng cân
      "W_AG1_KL.BRO" : Real;   // Phễu cân Cốt liệu 1_Khối lượng báo rỗng
      "W_AG1_KL.RUG" : Real;   // Phễu cân Cốt liệu 1_Khối lượng rung cân
      "W_AG1_TG.ON_RUNG" : Real;   // Phễu cân Cốt liệu 1_Thời gian bật rung
      "W_AG1_TG.OF_RUNG" : Real;   // Phễu cân Cốt liệu 1_Thời gian tắt rung
      "W_FD1_TG.DLC" : Real;   // Phễu cân FD 1_Thời gian trễ cân
      "W_FD1_TG.DLX" : Real;   // Phễu cân FD 1_Thời gian trễ xả
      "W_FD1_TG.DLD" : Real;   // Phễu cân FD 1_Thời gian trễ đóng cân
      "W_FD1_KL.BRO" : Real;   // Phễu cân FD 1_Khối lượng báo rỗng
      "W_FD1_KL.RUG" : Real;   // Phễu cân FD1_Khối lượng rung cân
      "W_FD1_TG.ON_RUNG" : Real;   // Phễu cân FD 1_Thời gian bật rung
      "W_FD1_TG.OF_RUNG" : Real;   // Phễu cân FD 1_Thời gian tắt rung
      "W_AP1_TG.DLC" : Real;   // Phễu cân Nhựa 1_Thời gian trễ cân
      "W_AP1_TG.DLX" : Real;   // Phễu cân Nhựa 1_Thời gian trễ xả
      "W_AP1_TG.DLD" : Real;   // Phễu cân Nhựa 1_Thời gian trễ đóng cân
      "W_AP1_KL.BRO" : Real;   // Phễu cân Nhựa 1_Khối lượng báo rỗng
      "W_SB1_TG.DLC" : Real;   // Phễu cân SBS 1_Thời gian trễ cân
      "W_SB1_TG.DLX" : Real;   // Phễu cân SBS 1_Thời gian trễ xả
      "W_SB1_TG.DLD" { ExternalWritable := 'False'} : Real;   // Phễu cân SBS 1_Thời gian trễ đóng cân
      "W_SB1_KL.BRO" : Real;   // Phễu cân SBS 1_Khối lượng báo rỗng
      "W_SB1_KL.RUG" : Real;   // Phễu cân SBS 1_Khối lượng rung cân
      "W_SB1_TG.ON_RUNG" : Real;   // Phễu cân SBS 1_Thời gian bật rung
      "W_SB1_TG.OF_RUNG" : Real;   // Phễu cân SBS 1_Thời gian tắt rung
      SO_ME_TRON : Real;   // Số mẻ cần trộn
      SV_AG1 : Real;   // Khối lượng Cần cân Cốt liệu 1
      SV_AG2 : Real;   // Khối lượng Cần cân Cốt liệu 2
      SV_AG3 : Real;   // Khối lượng Cần cân Cốt liệu 3
      SV_AG4 : Real;   // Khối lượng Cần cân Cốt liệu 4
      SV_AG5 : Real;   // Khối lượng Cần cân Cốt liệu 5
      SV_FD1 : Real;   // Khối lượng Cần cân FD 1
      SV_AP1 : Real;   // Khối lượng Cần cân Nhựa 1
      SV_SB1 : Real;   // Khối lượng Cần cân SBS 1
   END_VAR
BEGIN
END_DATA_BLOCK

DATA_BLOCK "C#5_WD_TIMER"   // DB5
{ S7_Optimized_Access := 'FALSE' }
VERSION : 0.1
// stored: AutoNumber true, CodeModifiedDate 2024-09-25T16:11:16.0895396Z, CompileDate 2025-08-30T17:40:34.4162196Z, CreationDate 2024-10-12T12:36:08.0193576Z, DBAccessibleFromOPCUA true, InterfaceModifiedDate 2024-09-25T16:11:16.0895396Z, IsConsistent true, IsKnowHowProtected false, IsOnlyStoredInLoadMemory false, IsPLCDB false, IsWriteProtectedInAS false, ModifiedDate 2024-10-13T07:10:46.0630795Z, ParameterModified 2024-09-25T16:11:16.0895396Z, StructureModified 2024-09-25T16:11:16.0895396Z
   VAR RETAIN
      TG_Tron : Real;   // Thời gian trộn
      TG_Xa100 : Real;   // Thời gian mở cửa nồi 100
      "TG_Xa FD Sau AG" : Real;   // Thời gian xả FD sau AG
      "TG_Xa AP Sau AG" : Real;   // Thời gian xả AP sau AG
      "TG_Xa SBS Sau AG" : Real;   // Thời gian xả SBS sau AG
      "TG_Bom Tuoi Nhua" : Real;   // Thời gian bơm tưới nhựa chạy thêm
      HSN_AG1 : Real;   // Hệ số nạp mô phỏng AG1
      HSN_AG2 : Real;   // Hệ số nạp mô phỏng AG2
      HSN_AG3 : Real;   // Hệ số nạp mô phỏng AG3
      HSN_AG4 : Real;   // Hệ số nạp mô phỏng AG4
      HSN_AG5 : Real;   // Hệ số nạp mô phỏng AG5
      HSX_AG1 : Real;   // Hệ số xả mô phỏng AG1
      HSN_FD1 : Real;   // Hệ số nạp mô phỏng FD1
      HSX_FD1 : Real;   // Hệ số xả mô phỏng FD1
      HSN_AP1 : Real;   // Hệ số nạp mô phỏng AP1
      HSX_AP1 : Real;   // Hệ số xả mô phỏng AP1
      HSN_SB1 : Real;   // Hệ số nạp mô phỏng SBS1
      HSX_SB1 : Real;   // Hệ số xả mô phỏng SBS1
   END_VAR
BEGIN
END_DATA_BLOCK

DATA_BLOCK "C#6_WD_CALIB"   // DB6
{ S7_Optimized_Access := 'FALSE' }
VERSION : 0.1
// stored: AutoNumber true, CodeModifiedDate 2026-01-01T14:21:06.6662125Z, CompileDate 2026-01-04T03:21:25.721467Z, CreationDate 2024-10-12T12:36:08.0193576Z, DBAccessibleFromOPCUA true, InterfaceModifiedDate 2026-01-01T14:21:06.6662125Z, IsConsistent true, IsKnowHowProtected false, IsOnlyStoredInLoadMemory false, IsPLCDB false, IsWriteProtectedInAS false, ModifiedDate 2026-01-01T14:21:06.6662125Z, ParameterModified 2026-01-01T14:21:06.6662125Z, StructureModified 2026-01-01T14:21:06.6662125Z
   VAR RETAIN
      KL_ZERO_AG1 : Real;   // Khối lượng chỉnh 0 cân AG1
      KL_SPAN_AG1 : Real;   // Khối lượng chỉnh tải cân AG1
      KL_ZERO_FD1 : Real;   // Khối lượng chỉnh 0 cân FD1
      KL_SPAN_FD1 : Real;   // Khối lượng chỉnh tải cân FD1
      KL_ZERO_AP1 : Real;   // Khối lượng chỉnh 0 cân AP1
      KL_SPAN_AP1 : Real;   // Khối lượng chỉnh tải cân AP1
      KL_ZERO_SB1 : Real;   // Khối lượng chỉnh 0 cân SB1
      KL_SPAN_SB1 : Real;   // Khối lượng chỉnh tải cân SB1
      ZERO_TEMP_TS : Real;   // Nhiệt độ T1 tan sấy
      SPAN_TEMP_TS : Real;   // Nhiệt độ T2 tan sấy
      ZERO_TEMP_AG : Real;   // Nhiệt độ T1 Cốt liệu Agg
      SPAN_TEMP_AG : Real;   // Nhiệt độ T2 Cốt kiệu Agg
      ZERO_TEMP_AP : Real;   // Nhiệt độ T1 Nhựa
      SPAN_TEMP_AP : Real;   // Nhiệt độ T2 Nhựa
      ZERO_TEMP_TL : Real;   // Nhiệt độ T1 Túi lọc
      SPAN_TEMP_TL : Real;   // Nhiệt độ T2 Túi lọc
      HS_AG1 : Real;   // Hệ số cân Ag1
      HS_FD1 : Real;   // Hệ số cân FD1
      HS_AP1 : Real;   // Hệ số cân AP1
      HS_SB1 : Real;   // Hệ số cân SB1
      "HS_TEMP TS" : Real;   // Hệ số nhiệt độ 1
      "HS_TEMP AG" : Real;   // Hệ số nhiệt độ 2
      "HS_TEMP AP" : Real;   // Hệ số nhiệt độ 3
      "HS_TEMP TL" : Real;   // Hệ số nhiệt độ 4
      XUNG_AG1 : Real;   // Đọc xung AG1
      XUNG_FD1 : Real;   // Đọc xung FD1
      XUNG_AP1 : Real;   // Đọc xung AP1
      XUNG_SB1 : Real;   // Đọc xung SB1
      XUNG_TEMP_TS : Real;   // Đọc xung nhiệt độ tan sấy
      XUNG_TEMP_AG : Real;   // Đọc xung nhiệt độ AGG
      XUNG_TEMP_AP : Real;   // Đọc xung nhiệt độ nhựa
      XUNG_TEMP_TL : Real;   // Đọc xung nhiệt độ túi lọc
      KLT_AG1 : Real;   // Đọc khối lượng cân AG
      KLT_FD1 : Real;   // Đọc khối lượng cân FD
      KLT_AP1 : Real;   // Đọc khối lượng cân AP
      KLT_SB1 : Real;   // Đọc khối lượng cân SBS
      NDT_TS : Real;   // Đọc nhiệt độ tan sấy
      NDT_AG : Real;   // Đọc nhiệt độ cốt liệu
      NDT_AP : Real;   // Đọc nhiệt độ nhựa
      NDT_TL : Real;   // Đọc nhiệt độ túi lọc bụi
      HMI_Manual_Pulse : Bool;
      KL_ZERO_IND_AGG1 : Real;
      KL_SPAN_IND_AGG1 : Real;
      HS_IND_AGG1 : Real;
      XUNG_IND_AGG1 : Real;
      KLT_IND_AGG1 : Real;
      KL_ZERO_IND_AGG2 : Real;
      KL_SPAN_IND_AGG2 : Real;
      HS_IND_AGG2 : Real;
      XUNG_IND_AGG2 : Real;
      KLT_IND_AGG2 : Real;
      KL_ZERO_IND_AGG3 : Real;
      KL_SPAN_IND_AGG3 : Real;
      HS_IND_AGG3 : Real;
      XUNG_IND_AGG3 : Real;
      KLT_IND_AGG3 : Real;
      KL_ZERO_IND_AGG4 : Real;
      KL_SPAN_IND_AGG4 : Real;
      HS_IND_AGG4 : Real;
      XUNG_IND_AGG4 : Real;
      KLT_IND_AGG4 : Real;
      KL_ZERO_IND_AGG5 : Real;
      KL_SPAN_IND_AGG5 : Real;
      HS_IND_AGG5 : Real;
      XUNG_IND_AGG5 : Real;
      KLT_IND_AGG5 : Real;
   END_VAR
BEGIN
END_DATA_BLOCK

DATA_BLOCK "C#7_RD_RUN"   // DB7
{ S7_Optimized_Access := 'FALSE' }
VERSION : 0.1
// stored: AutoNumber true, CodeModifiedDate 2024-10-13T07:13:35.9743236Z, CompileDate 2025-08-30T17:40:32.1468413Z, CreationDate 2024-10-12T12:36:08.0193576Z, DBAccessibleFromOPCUA true, InterfaceModifiedDate 2024-10-13T07:13:35.9743236Z, IsConsistent true, IsKnowHowProtected false, IsOnlyStoredInLoadMemory false, IsPLCDB false, IsWriteProtectedInAS false, ModifiedDate 2024-10-13T07:14:11.4381467Z, ParameterModified 2024-10-13T07:13:35.9743236Z, StructureModified 2024-10-13T07:13:35.9743236Z
   VAR RETAIN
      PV_AG1 : Real;   // Thực cân cốt liệu 1
      "%_WAG1" : Real;   // Phần trăm khối lượng cốt liệu 1
      WE_AG1 : Real;   // Khối lượng cân cốt liệu 1
      SMC_AG1 : Real;   // Số mẻ cân phễu cân cốt liệu 1
      SMX_AG1 : Real;   // Số mẻ xả phễu cân cốt liệu 1
      PV_AG2 : Real;   // Thực cân cốt liệu 2
      SMC_AG2 : Real;   // Số mẻ cân phễu cân cốt liệu 2
      SMX_AG2 : Real;   // Số mẻ xả phễu cân cốt liệu 2
      PV_AG3 : Real;   // Thực cân cốt liệu 3
      SMC_AG3 : Real;   // Số mẻ cân phễu cân cốt liệu 3
      SMX_AG3 : Real;   // Số mẻ xả phễu cân cốt liệu 3
      PV_AG4 : Real;   // Thực cân cốt liệu 4
      SMC_AG4 : Real;   // Số mẻ cân phễu cân cốt liệu 4
      SMX_AG4 : Real;   // Số mẻ xả phễu cân cốt liệu 4
      PV_AG5 : Real;   // Thực cân cốt liệu 5
      SMC_AG5 : Real;   // Số mẻ cân phễu cân cốt liệu 5
      SMX_AG5 : Real;   // Số mẻ xả phễu cân cốt liệu 5
      PV_FD1 : Real;   // Thực cân silo FD 1
      "%_WFD1" : Real;   // Phần trăm khối lượng phễu cân FD 1
      WE_FD1 : Real;   // Khối lượng phễu cân FD 1
      SMC_FD1 : Real;   // Số mẻ cân phễu cân FD 1
      SMX_FD1 : Real;   // Số mẻ xả phễu cân FD 1
      PV_AP1 : Real;   // Thực cân Nhựa 1
      "%_WAP1" : Real;   // Phần trăm khối lượng phễu cân Nhựa 1
      WE_AP1 : Real;   // Khối lượng phễu cân Nhựa 1
      SMC_AP1 : Real;   // Số mẻ cân phễu cân Nhựa 1
      SMX_AP1 : Real;   // Số mẻ xả phễu cân Nhựa 1
      PV_SB1 : Real;   // Thực cân SBS 1
      "%_WSB1" : Real;   // Phần trăm khối lượng phễu cân SBS 1
      WE_SB1 : Real;   // Khối lượng phễu cân SBS 1
      SMC_SB1 : Real;   // Số mẻ cân phễu cân SBS 1
      SMX_SB1 : Real;   // Số mẻ xả phễu cân SBS 1
      SMC_MIXER : Real;   // Số mẻ cân nồi trộn
      SMX_MIXER : Real;   // Số mẻ xả nồi trộn
      "TG_THUC TRON" : Real;   // Thoi gian thuc tron
      TG_THUC_XA : Real;   // Thoi gian thuc xa
      SMT : Real;
      "M3/ME" : Real;
      PVM_AG1 : Real;   // Thực cân tay cốt liệu 1
      PVM_AG2 : Real;   // Thực cân tay cốt liệu 2
      PVM_AG3 : Real;   // Thực cân tay cốt liệu 3
      PVM_AG4 : Real;   // Thực cân tay cốt liệu 4
      PVM_AG5 : Real;   // Thực cân tay cốt liệu 5
      PVM_FD1 : Real;   // Thực cân tay FD1
      PVM_AP1 : Real;   // Thực cân tay Nhựa
      PVM_SB1 : Real;   // Thực cân tay SBS1
      TEMP_TUILOC : Real;   // Nhiệt độ túi lọc hiển thị
      TEMP_AGG : Real;   // Nhiệt độ cốt liệu hiển thị
      TEMP_TANSAY : Real;   // Nhiệt độ tan sấy hiển thị
      TEMP_NHUA : Real;   // Nhiệt độ nhựa hiển thị
   END_VAR
BEGIN
END_DATA_BLOCK

DATA_BLOCK "C#8_RD_REPORT"   // DB8
{ S7_Optimized_Access := 'FALSE' }
VERSION : 0.1
// stored: AutoNumber false, CodeModifiedDate 2024-09-25T16:49:35.7764199Z, CompileDate 2025-08-30T17:40:31.7117876Z, CreationDate 2024-10-12T12:36:08.0193576Z, DBAccessibleFromOPCUA true, InterfaceModifiedDate 2024-09-25T16:49:35.7764199Z, IsConsistent true, IsKnowHowProtected false, IsOnlyStoredInLoadMemory false, IsPLCDB false, IsWriteProtectedInAS false, ModifiedDate 2024-10-13T07:15:20.7288707Z, ParameterModified 2024-09-25T16:49:35.7764199Z, StructureModified 2024-09-25T16:49:35.7764199Z
   VAR
      SAVE_REPORT : Bool;   // Lưu dữ liệu trộn
      SAVE_REPORT_1 : Bool;
      SAVE_REPORT_2 : Bool;
      SAVE_REPORT_3 : Bool;
      SAVE_REPORT_4 : Bool;
      SAVE_REPORT_5 : Bool;
      SAVE_REPORT_6 : Bool;
      SAVE_REPORT_7 : Bool;
      SAVE_REPORT_8 : Bool;
      SAVE_REPORT_9 : Bool;
      SAVE_REPORT_10 : Bool;
      SAVE_REPORT_11 : Bool;
      SAVE_REPORT_12 : Bool;
      SAVE_REPORT_13 : Bool;
      SAVE_REPORT_14 : Bool;
      SAVE_REPORT_15 : Bool;
      SAVE_REPORT_16 : Bool;
      PV_AGG1 : Real;   // Thực cân Cốt liệu 1
      PVM_AGG1 : Real;   // Cân tay Cốt liệu 1
      PV_AGG2 : Real;   // Thực cân Cốt liệu 2
      PVM_AGG2 : Real;   // Cân tay Cốt liệu 2
      PV_AGG3 : Real;   // Thực cân Cốt liệu 3
      PVM_AGG3 : Real;   // Cân tay Cốt liệu 3
      PV_AGG4 : Real;   // Thực cân Cốt liệu 4
      PVM_AGG4 : Real;   // Cân tay Cốt liệu 4
      PV_AGG5 : Real;   // Thực cân Cốt liệu 5
      PVM_AGG5 : Real;   // Cân tay Cốt liệu 5
      TEMP_TS : Real;   // Nhiệt độ tang sấy
      TEMP_AG : Real;   // Nhiệt độ cốt liệu
      PV_FD1 : Real;   // Thực cân F/D 1
      PVM_FD1 : Real;   // Cân tay F/D 1
      PV_AP1 : Real;   // Thực cân Nhựa 1
      PVM_AP1 : Real;   // Cân tay Nhựa 1
      TEMP_AP : Real;   // Nhiệt độ nhựa
      PV_SB1 : Real;   // Thực cân SBS 1
      PVM_SB1 : Real;   // Cân tay SBS 1
   END_VAR
BEGIN
END_DATA_BLOCK

DATA_BLOCK "PLC_BIT"   // DB9
{ S7_Optimized_Access := 'FALSE' }
VERSION : 0.1
// stored: AutoNumber true, CodeModifiedDate 2026-01-01T12:46:58.5268647Z, CompileDate 2026-01-01T12:47:15.7550826Z, CreationDate 2024-10-12T12:36:08.0193576Z, DBAccessibleFromOPCUA true, InterfaceModifiedDate 2026-01-01T12:46:58.5268647Z, IsConsistent true, IsKnowHowProtected false, IsOnlyStoredInLoadMemory false, IsPLCDB false, IsWriteProtectedInAS false, ModifiedDate 2026-01-01T12:46:58.5268647Z, ParameterModified 2026-01-01T12:46:58.5268647Z, StructureModified 2026-01-01T12:46:58.5268647Z
   VAR
      RUN : Bool;
      MAN : Bool;
      AUT : Bool;
      SIM : Bool;
      PAU : Bool;
      NTR_FU : Bool;
      PCH_FU : Bool;
      SKIP_FU : Bool;
      AGG1_FU : Bool;
      WAG1_FU : Bool;
      WAG1_EM : Bool;
      AGG2_FU : Bool;
      WAG2_FU : Bool;
      WAG2_EM : Bool;
      AGG3_FU : Bool;
      WAG3_FU : Bool;
      WAG3_EM : Bool;
      AGG4_FU : Bool;
      WAG4_FU : Bool;
      WAG4_EM : Bool;
      AGG5_FU : Bool;
      WAG5_FU : Bool;
      WAG5_EM : Bool;
      AGG6_FU : Bool;
      WAG6_FU : Bool;
      WAG6_EM : Bool;
      CEM1_FU : Bool;
      CEM2_FU : Bool;
      CEM3_FU : Bool;
      WCE1_FU : Bool;
      WCE1_EM : Bool;
      CEM4_FU : Bool;
      CEM5_FU : Bool;
      WCE2_FU : Bool;
      WCE2_EM : Bool;
      WAT1_FU : Bool;
      WWA1_FU : Bool;
      WWA1_EM : Bool;
      WAT2_FU : Bool;
      WWA2_FU : Bool;
      WWA2_EM : Bool;
      ADD1_FU : Bool;
      ADD2_FU : Bool;
      ADD3_FU : Bool;
      WAD1_FU : Bool;
      WAD1_EM : Bool;
      ADD4_FU : Bool;
      ADD5_FU : Bool;
      ADD6_FU : Bool;
      WAD2_FU : Bool;
      WAD2_EM : Bool;
      "BAT/TAT NT" : Bool;
      "BAT/TAT BTX" : Bool;
      "NN_CAN NUOC" : Bool;
      "NN_XA NUOC" : Bool;
      NN_MCN : Bool;
      NN_DCN : Bool;
      "NN_DONG KEP" : Bool;
      "NN_MO KEP" : Bool;
      "NN_GAU LEN" : Bool;
      "NN_DUNG GAU" : Bool;
      "NN_GAU XUONG" : Bool;
      TOP_BTC : Bool;
      "TOP. GAU LEN" : Bool;
      "TOP. GAU XUONG" : Bool;
      "COT LIEU_FU" : Bool;
      PCĐ_SIM : Bool;
      PCM_SIM : Bool;
      CNĐ_SIM : Bool;
      CNM_SIM : Bool;
      "CN1/2_SIM" : Bool;
      COT_LIEU_FU : Bool;
      KT_XA_AGG : Bool;
      NEXT_WAGG1 : Bool;
      NEXT_WAGG2 : Bool;
      NEXT_WAGG3 : Bool;
      NEXT_WAGG4 : Bool;
      NEXT_WAGG5 : Bool;
      NEXT_WAGG6 : Bool;
      NEXT_WCEM1 : Bool;
      NEXT_WCEM2 : Bool;
      NEXT_WWAT1 : Bool;
      NEXT_WWAT2 : Bool;
      NEXT_WADD1 : Bool;
      NEXT_WADD2 : Bool;
      End_Agg1 : Bool;
      End_Agg2 : Bool;
      End_Agg3 : Bool;
      End_Agg4 : Bool;
      End_Agg5 : Bool;
      End_Agg6 : Bool;
      SW_MODE : Bool;
   END_VAR
BEGIN
END_DATA_BLOCK

DATA_BLOCK "PLC_DATA"   // DB10
{ S7_Optimized_Access := 'FALSE' }
VERSION : 0.1
// stored: AutoNumber true, CodeModifiedDate 2026-01-04T14:16:44.6751265Z, CompileDate 2026-01-04T14:27:04.9564115Z, CreationDate 2024-10-12T12:36:08.0193576Z, DBAccessibleFromOPCUA true, InterfaceModifiedDate 2026-01-04T14:16:44.6751265Z, IsConsistent true, IsKnowHowProtected false, IsOnlyStoredInLoadMemory false, IsPLCDB false, IsWriteProtectedInAS false, ModifiedDate 2026-01-04T14:16:44.6751265Z, ParameterModified 2026-01-04T14:16:44.6751265Z, StructureModified 2026-01-04T14:16:44.6751265Z
   VAR RETAIN
      SI_WAG : Real;
      RE_WAG : Real;
      SI_WFD : Real;
      RE_WFD : Real;
      SI_WAP : Real;
      RE_WAP : Real;
      SI_WSB : Real;
      RE_WSB : Real;
      TEMP_TL : DInt;
      TEMP_TS : DInt;
      TEMP_AG : DInt;
      TEMP_AP : DInt;
      TG_TRON : Real;
      TG_XA : Real;
      M3_MAX : Real;
      SMC_SILO_AG1 : Real;
      SMC_SILO_AG2 : Real;
      SMC_SILO_AG3 : Real;
      SMC_SILO_AG4 : Real;
      SMC_SILO_AG5 : Real;
      SMC_SILO_FD1 : Real;
      SMC_SILO_AP1 : Real;
      SMC_SILO_SB1 : Real;
      SI_WAGG1 : Real;
      RE_WAGG1 : Real;
      SI_WAGG2 : Real;
      RE_WAGG2 : Real;
      SI_WAGG3 : Real;
      RE_WAGG3 : Real;
      SI_WAGG4 : Real;
      RE_WAGG4 : Real;
      SI_WAGG5 : Real;
      RE_WAGG5 : Real;
   END_VAR
BEGIN
END_DATA_BLOCK

ORGANIZATION_BLOCK "Main_P1"   // OB1, LAD, ProgramCycle
TITLE = "Main Program Sweep (Cycle)"
{ S7_Optimized_Access := 'TRUE' }
VERSION : 0.1
// stored: AutoNumber true, CodeModifiedDate 2026-01-04T14:29:42.3003179Z, CompileDate 2026-01-04T14:29:49.7688293Z, ConstantName OB_Main_P1, CreationDate 2024-10-12T12:36:08.0193576Z, EventClass Program cycle, HandleErrorsWithinBlock false, InterfaceModifiedDate 2008-07-21T16:55:08.419547Z, IsConsistent true, IsIECCheckEnabled false, IsKnowHowProtected false, IsWriteProtected false, ModifiedDate 2026-01-04T14:29:42.3003179Z, ParameterModified 2008-07-21T16:55:08.419547Z, PLCSimAdvancedSupport false, PriorityNumber 1, ProcessImagePartNumber 65535, SetENOAutomatically False, StructureModified 2008-07-21T16:55:08.419547Z
   VAR_INPUT
      Initial_Call : Bool;   // Initial call of this OB
      Remanence : Bool;   // =True, if remanent data are available
   END_VAR
   VAR_TEMP   // added for the SCL form of the ladder/FBD networks
      _w1 : Bool;
      _w2 : Bool;
      _w3 : Bool;
      _w4 : Bool;
      _w5 : Bool;
      _w6 : Bool;
   END_VAR
BEGIN

REGION Network 1: MOVE INPUT
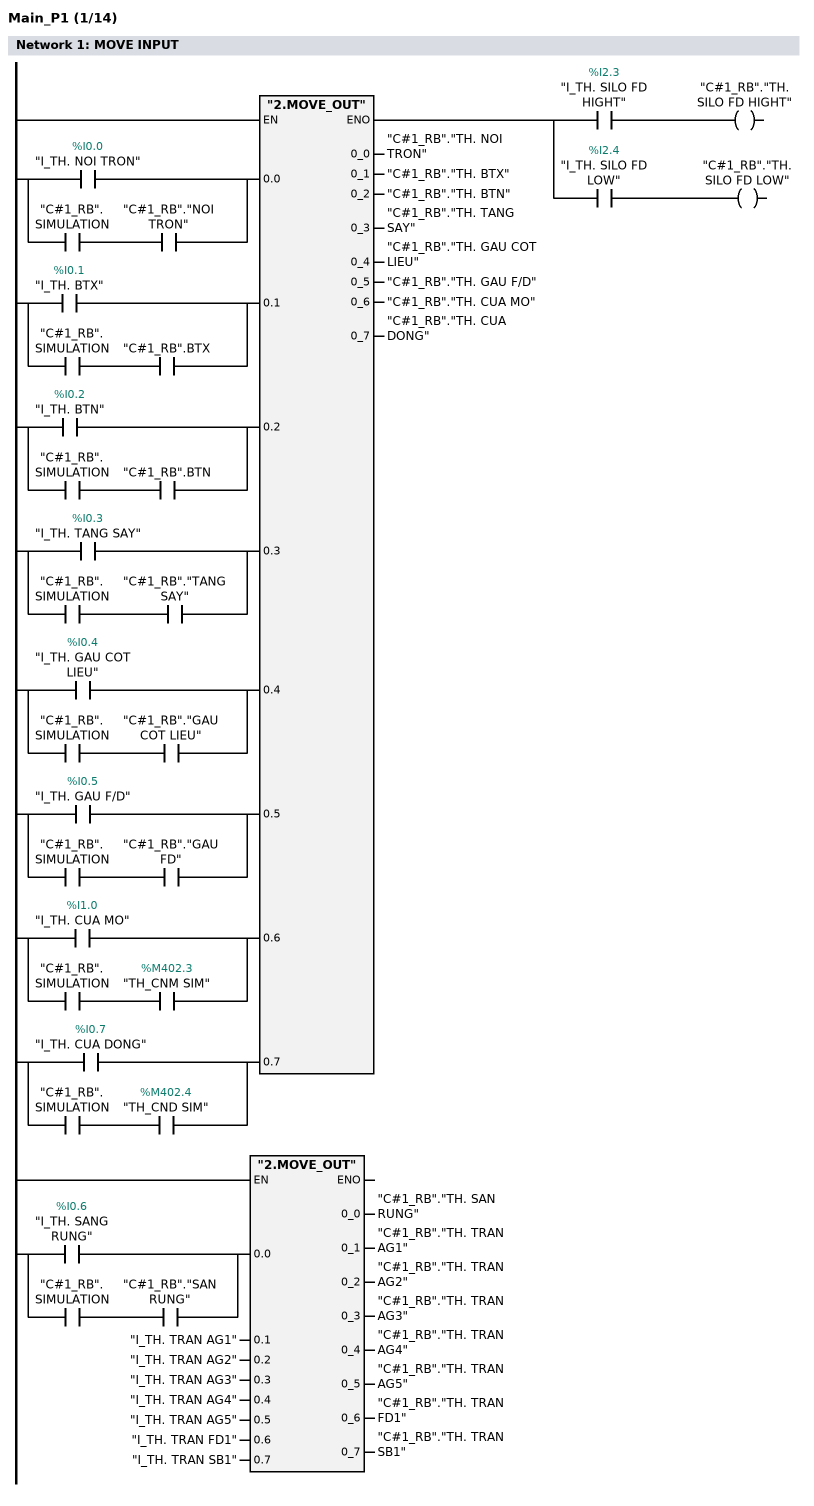
   RUNG wire#powerrail
      "2.MOVE_OUT"("0.0" := wire#w1, "0.1" := wire#w2, "0.2" := wire#w3, "0.3" := wire#w4, "0.4" := wire#w5, "0.5" := wire#w6, "0.6" := wire#w7, "0.7" := wire#w8, "0_0" => "C#1_RB"."TH. NOI TRON", "0_1" => "C#1_RB"."TH. BTX", "0_2" => "C#1_RB"."TH. BTN", "0_3" => "C#1_RB"."TH. TANG SAY", "0_4" => "C#1_RB"."TH. GAU COT LIEU", "0_5" => "C#1_RB"."TH. GAU F/D", "0_6" => "C#1_RB"."TH. CUA MO", "0_7" => "C#1_RB"."TH. CUA DONG")
      wire#w9
      Contact( "I_TH. SILO FD HIGHT" )
      Coil( "C#1_RB"."TH. SILO FD HIGHT" )
   END_RUNG
   RUNG wire#powerrail
      Contact( "I_TH. NOI TRON" )
   END_RUNG wire#w1
   RUNG wire#powerrail
      Contact( "C#1_RB".SIMULATION )
      Contact( "C#1_RB"."NOI TRON" )
   END_RUNG wire#w1
   RUNG wire#powerrail
      Contact( "I_TH. BTX" )
   END_RUNG wire#w2
   RUNG wire#powerrail
      Contact( "C#1_RB".SIMULATION )
      Contact( "C#1_RB".BTX )
   END_RUNG wire#w2
   RUNG wire#powerrail
      Contact( "I_TH. BTN" )
   END_RUNG wire#w3
   RUNG wire#powerrail
      Contact( "C#1_RB".SIMULATION )
      Contact( "C#1_RB".BTN )
   END_RUNG wire#w3
   RUNG wire#powerrail
      Contact( "I_TH. TANG SAY" )
   END_RUNG wire#w4
   RUNG wire#powerrail
      Contact( "C#1_RB".SIMULATION )
      Contact( "C#1_RB"."TANG SAY" )
   END_RUNG wire#w4
   RUNG wire#powerrail
      Contact( "I_TH. GAU COT LIEU" )
   END_RUNG wire#w5
   RUNG wire#powerrail
      Contact( "C#1_RB".SIMULATION )
      Contact( "C#1_RB"."GAU COT LIEU" )
   END_RUNG wire#w5
   RUNG wire#powerrail
      Contact( "I_TH. GAU F/D" )
   END_RUNG wire#w6
   RUNG wire#powerrail
      Contact( "C#1_RB".SIMULATION )
      Contact( "C#1_RB"."GAU FD" )
   END_RUNG wire#w6
   RUNG wire#powerrail
      Contact( "I_TH. CUA MO" )
   END_RUNG wire#w7
   RUNG wire#powerrail
      Contact( "C#1_RB".SIMULATION )
      Contact( "TH_CNM SIM" )
   END_RUNG wire#w7
   RUNG wire#powerrail
      Contact( "I_TH. CUA DONG" )
   END_RUNG wire#w8
   RUNG wire#powerrail
      Contact( "C#1_RB".SIMULATION )
      Contact( "TH_CND SIM" )
   END_RUNG wire#w8
   RUNG wire#w9
      Contact( "I_TH. SILO FD LOW" )
      Coil( "C#1_RB"."TH. SILO FD LOW" )
   END_RUNG
   RUNG wire#powerrail
      "2.MOVE_OUT"("0.0" := wire#w10, "0.1" := "I_TH. TRAN AG1", "0.2" := "I_TH. TRAN AG2", "0.3" := "I_TH. TRAN AG3", "0.4" := "I_TH. TRAN AG4", "0.5" := "I_TH. TRAN AG5", "0.6" := "I_TH. TRAN FD1", "0.7" := "I_TH. TRAN SB1", "0_0" => "C#1_RB"."TH. SAN RUNG", "0_1" => "C#1_RB"."TH. TRAN AG1", "0_2" => "C#1_RB"."TH. TRAN AG2", "0_3" => "C#1_RB"."TH. TRAN AG3", "0_4" => "C#1_RB"."TH. TRAN AG4", "0_5" => "C#1_RB"."TH. TRAN AG5", "0_6" => "C#1_RB"."TH. TRAN FD1", "0_7" => "C#1_RB"."TH. TRAN SB1")
   END_RUNG
   RUNG wire#powerrail
      Contact( "I_TH. SANG RUNG" )
   END_RUNG wire#w10
   RUNG wire#powerrail
      Contact( "C#1_RB".SIMULATION )
      Contact( "C#1_RB"."SAN RUNG" )
   END_RUNG wire#w10
   // the same network as SCL:
   "2.MOVE_OUT"("0.0" := "I_TH. NOI TRON" OR ("C#1_RB".SIMULATION AND "C#1_RB"."NOI TRON"),
                "0.1" := "I_TH. BTX" OR ("C#1_RB".SIMULATION AND "C#1_RB".BTX),
                "0.2" := "I_TH. BTN" OR ("C#1_RB".SIMULATION AND "C#1_RB".BTN),
                "0.3" := "I_TH. TANG SAY" OR ("C#1_RB".SIMULATION AND "C#1_RB"."TANG SAY"),
                "0.4" := "I_TH. GAU COT LIEU" OR ("C#1_RB".SIMULATION AND "C#1_RB"."GAU COT LIEU"),
                "0.5" := "I_TH. GAU F/D" OR ("C#1_RB".SIMULATION AND "C#1_RB"."GAU FD"),
                "0.6" := "I_TH. CUA MO" OR ("C#1_RB".SIMULATION AND "TH_CNM SIM"),
                "0.7" := "I_TH. CUA DONG" OR ("C#1_RB".SIMULATION AND "TH_CND SIM"),
                "0_0" => "C#1_RB"."TH. NOI TRON",
                "0_1" => "C#1_RB"."TH. BTX",
                "0_2" => "C#1_RB"."TH. BTN",
                "0_3" => "C#1_RB"."TH. TANG SAY",
                "0_4" => "C#1_RB"."TH. GAU COT LIEU",
                "0_5" => "C#1_RB"."TH. GAU F/D",
                "0_6" => "C#1_RB"."TH. CUA MO",
                "0_7" => "C#1_RB"."TH. CUA DONG",
                ENO => #_w1);
   "C#1_RB"."TH. SILO FD HIGHT" := #_w1 AND "I_TH. SILO FD HIGHT";
   "C#1_RB"."TH. SILO FD LOW" := #_w1 AND "I_TH. SILO FD LOW";
   "2.MOVE_OUT"("0.0" := "I_TH. SANG RUNG" OR ("C#1_RB".SIMULATION AND "C#1_RB"."SAN RUNG"),
                "0.1" := "I_TH. TRAN AG1",
                "0.2" := "I_TH. TRAN AG2",
                "0.3" := "I_TH. TRAN AG3",
                "0.4" := "I_TH. TRAN AG4",
                "0.5" := "I_TH. TRAN AG5",
                "0.6" := "I_TH. TRAN FD1",
                "0.7" := "I_TH. TRAN SB1",
                "0_0" => "C#1_RB"."TH. SAN RUNG",
                "0_1" => "C#1_RB"."TH. TRAN AG1",
                "0_2" => "C#1_RB"."TH. TRAN AG2",
                "0_3" => "C#1_RB"."TH. TRAN AG3",
                "0_4" => "C#1_RB"."TH. TRAN AG4",
                "0_5" => "C#1_RB"."TH. TRAN AG5",
                "0_6" => "C#1_RB"."TH. TRAN FD1",
                "0_7" => "C#1_RB"."TH. TRAN SB1");
END_REGION

REGION Network 2: MOVE OUTPUT
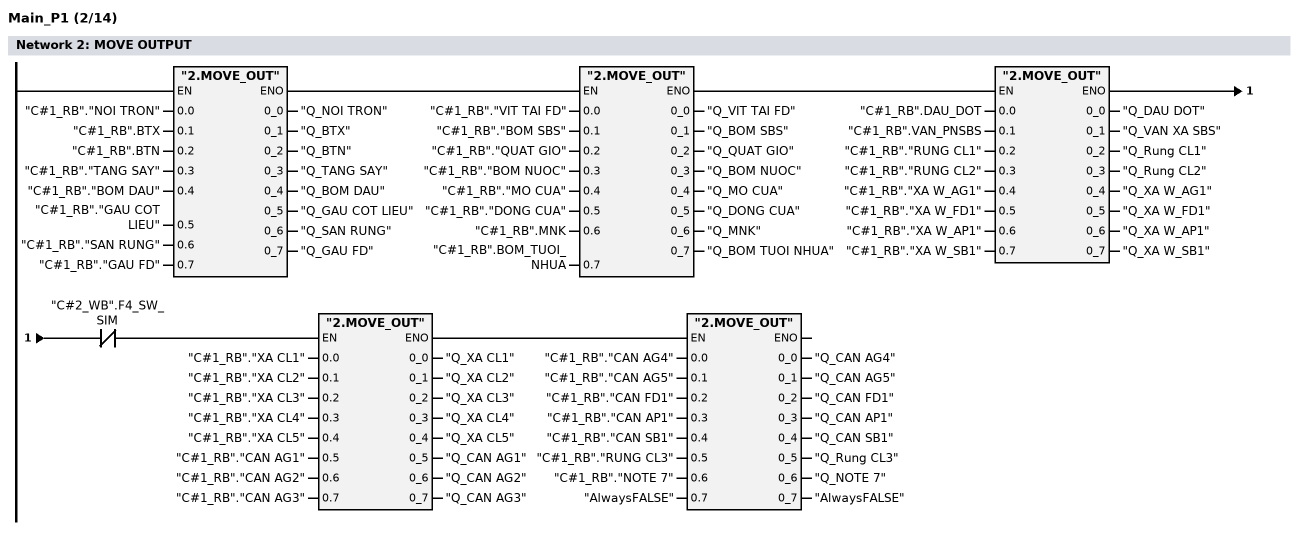
   RUNG wire#powerrail
      "2.MOVE_OUT"("0.0" := "C#1_RB"."NOI TRON", "0.1" := "C#1_RB".BTX, "0.2" := "C#1_RB".BTN, "0.3" := "C#1_RB"."TANG SAY", "0.4" := "C#1_RB"."BOM DAU", "0.5" := "C#1_RB"."GAU COT LIEU", "0.6" := "C#1_RB"."SAN RUNG", "0.7" := "C#1_RB"."GAU FD", "0_0" => "Q_NOI TRON", "0_1" => "Q_BTX", "0_2" => "Q_BTN", "0_3" => "Q_TANG SAY", "0_4" => "Q_BOM DAU", "0_5" => "Q_GAU COT LIEU", "0_6" => "Q_SAN RUNG", "0_7" => "Q_GAU FD")
      "2.MOVE_OUT"("0.0" := "C#1_RB"."VIT TAI FD", "0.1" := "C#1_RB"."BOM SBS", "0.2" := "C#1_RB"."QUAT GIO", "0.3" := "C#1_RB"."BOM NUOC", "0.4" := "C#1_RB"."MO CUA", "0.5" := "C#1_RB"."DONG CUA", "0.6" := "C#1_RB".MNK, "0.7" := "C#1_RB".BOM_TUOI_NHUA, "0_0" => "Q_VIT TAI FD", "0_1" => "Q_BOM SBS", "0_2" => "Q_QUAT GIO", "0_3" => "Q_BOM NUOC", "0_4" => "Q_MO CUA", "0_5" => "Q_DONG CUA", "0_6" => "Q_MNK", "0_7" => "Q_BOM TUOI NHUA")
      "2.MOVE_OUT"("0.0" := "C#1_RB".DAU_DOT, "0.1" := "C#1_RB".VAN_PNSBS, "0.2" := "C#1_RB"."RUNG CL1", "0.3" := "C#1_RB"."RUNG CL2", "0.4" := "C#1_RB"."XA W_AG1", "0.5" := "C#1_RB"."XA W_FD1", "0.6" := "C#1_RB"."XA W_AP1", "0.7" := "C#1_RB"."XA W_SB1", "0_0" => "Q_DAU DOT", "0_1" => "Q_VAN XA SBS", "0_2" => "Q_Rung CL1", "0_3" => "Q_Rung CL2", "0_4" => "Q_XA W_AG1", "0_5" => "Q_XA W_FD1", "0_6" => "Q_XA W_AP1", "0_7" => "Q_XA W_SB1")
      I_Contact( "C#2_WB".F4_SW_SIM )
      "2.MOVE_OUT"("0.0" := "C#1_RB"."XA CL1", "0.1" := "C#1_RB"."XA CL2", "0.2" := "C#1_RB"."XA CL3", "0.3" := "C#1_RB"."XA CL4", "0.4" := "C#1_RB"."XA CL5", "0.5" := "C#1_RB"."CAN AG1", "0.6" := "C#1_RB"."CAN AG2", "0.7" := "C#1_RB"."CAN AG3", "0_0" => "Q_XA CL1", "0_1" => "Q_XA CL2", "0_2" => "Q_XA CL3", "0_3" => "Q_XA CL4", "0_4" => "Q_XA CL5", "0_5" => "Q_CAN AG1", "0_6" => "Q_CAN AG2", "0_7" => "Q_CAN AG3")
      "2.MOVE_OUT"("0.0" := "C#1_RB"."CAN AG4", "0.1" := "C#1_RB"."CAN AG5", "0.2" := "C#1_RB"."CAN FD1", "0.3" := "C#1_RB"."CAN AP1", "0.4" := "C#1_RB"."CAN SB1", "0.5" := "C#1_RB"."RUNG CL3", "0.6" := "C#1_RB"."NOTE 7", "0.7" := "AlwaysFALSE", "0_0" => "Q_CAN AG4", "0_1" => "Q_CAN AG5", "0_2" => "Q_CAN FD1", "0_3" => "Q_CAN AP1", "0_4" => "Q_CAN SB1", "0_5" => "Q_Rung CL3", "0_6" => "Q_NOTE 7", "0_7" => "AlwaysFALSE")
   END_RUNG
   // the same network as SCL:
   "2.MOVE_OUT"("0.0" := "C#1_RB"."NOI TRON",
                "0.1" := "C#1_RB".BTX,
                "0.2" := "C#1_RB".BTN,
                "0.3" := "C#1_RB"."TANG SAY",
                "0.4" := "C#1_RB"."BOM DAU",
                "0.5" := "C#1_RB"."GAU COT LIEU",
                "0.6" := "C#1_RB"."SAN RUNG",
                "0.7" := "C#1_RB"."GAU FD",
                "0_0" => "Q_NOI TRON",
                "0_1" => "Q_BTX",
                "0_2" => "Q_BTN",
                "0_3" => "Q_TANG SAY",
                "0_4" => "Q_BOM DAU",
                "0_5" => "Q_GAU COT LIEU",
                "0_6" => "Q_SAN RUNG",
                "0_7" => "Q_GAU FD",
                ENO => #_w1);
   "2.MOVE_OUT"(EN := #_w1,
                "0.0" := "C#1_RB"."VIT TAI FD",
                "0.1" := "C#1_RB"."BOM SBS",
                "0.2" := "C#1_RB"."QUAT GIO",
                "0.3" := "C#1_RB"."BOM NUOC",
                "0.4" := "C#1_RB"."MO CUA",
                "0.5" := "C#1_RB"."DONG CUA",
                "0.6" := "C#1_RB".MNK,
                "0.7" := "C#1_RB".BOM_TUOI_NHUA,
                "0_0" => "Q_VIT TAI FD",
                "0_1" => "Q_BOM SBS",
                "0_2" => "Q_QUAT GIO",
                "0_3" => "Q_BOM NUOC",
                "0_4" => "Q_MO CUA",
                "0_5" => "Q_DONG CUA",
                "0_6" => "Q_MNK",
                "0_7" => "Q_BOM TUOI NHUA",
                ENO => #_w2);
   "2.MOVE_OUT"(EN := #_w2,
                "0.0" := "C#1_RB".DAU_DOT,
                "0.1" := "C#1_RB".VAN_PNSBS,
                "0.2" := "C#1_RB"."RUNG CL1",
                "0.3" := "C#1_RB"."RUNG CL2",
                "0.4" := "C#1_RB"."XA W_AG1",
                "0.5" := "C#1_RB"."XA W_FD1",
                "0.6" := "C#1_RB"."XA W_AP1",
                "0.7" := "C#1_RB"."XA W_SB1",
                "0_0" => "Q_DAU DOT",
                "0_1" => "Q_VAN XA SBS",
                "0_2" => "Q_Rung CL1",
                "0_3" => "Q_Rung CL2",
                "0_4" => "Q_XA W_AG1",
                "0_5" => "Q_XA W_FD1",
                "0_6" => "Q_XA W_AP1",
                "0_7" => "Q_XA W_SB1",
                ENO => #_w3);
   "2.MOVE_OUT"(EN := #_w3 AND NOT "C#2_WB".F4_SW_SIM,
                "0.0" := "C#1_RB"."XA CL1",
                "0.1" := "C#1_RB"."XA CL2",
                "0.2" := "C#1_RB"."XA CL3",
                "0.3" := "C#1_RB"."XA CL4",
                "0.4" := "C#1_RB"."XA CL5",
                "0.5" := "C#1_RB"."CAN AG1",
                "0.6" := "C#1_RB"."CAN AG2",
                "0.7" := "C#1_RB"."CAN AG3",
                "0_0" => "Q_XA CL1",
                "0_1" => "Q_XA CL2",
                "0_2" => "Q_XA CL3",
                "0_3" => "Q_XA CL4",
                "0_4" => "Q_XA CL5",
                "0_5" => "Q_CAN AG1",
                "0_6" => "Q_CAN AG2",
                "0_7" => "Q_CAN AG3",
                ENO => #_w4);
   IF #_w4 THEN
       "2.MOVE_OUT"("0.0" := "C#1_RB"."CAN AG4",
                    "0.1" := "C#1_RB"."CAN AG5",
                    "0.2" := "C#1_RB"."CAN FD1",
                    "0.3" := "C#1_RB"."CAN AP1",
                    "0.4" := "C#1_RB"."CAN SB1",
                    "0.5" := "C#1_RB"."RUNG CL3",
                    "0.6" := "C#1_RB"."NOTE 7",
                    "0.7" := "AlwaysFALSE",
                    "0_0" => "Q_CAN AG4",
                    "0_1" => "Q_CAN AG5",
                    "0_2" => "Q_CAN FD1",
                    "0_3" => "Q_CAN AP1",
                    "0_4" => "Q_CAN SB1",
                    "0_5" => "Q_Rung CL3",
                    "0_6" => "Q_NOTE 7",
                    "0_7" => "AlwaysFALSE");
   END_IF;
END_REGION

REGION Network 3: ĐIỀU KHIỂN TAY
   // Nếu ở chế độ Tự động, mà TANG SẤY chưa được mở thì không bật được Băng tải xiêng, tương tự nếu chưa mở BTX thì không mở được BTN
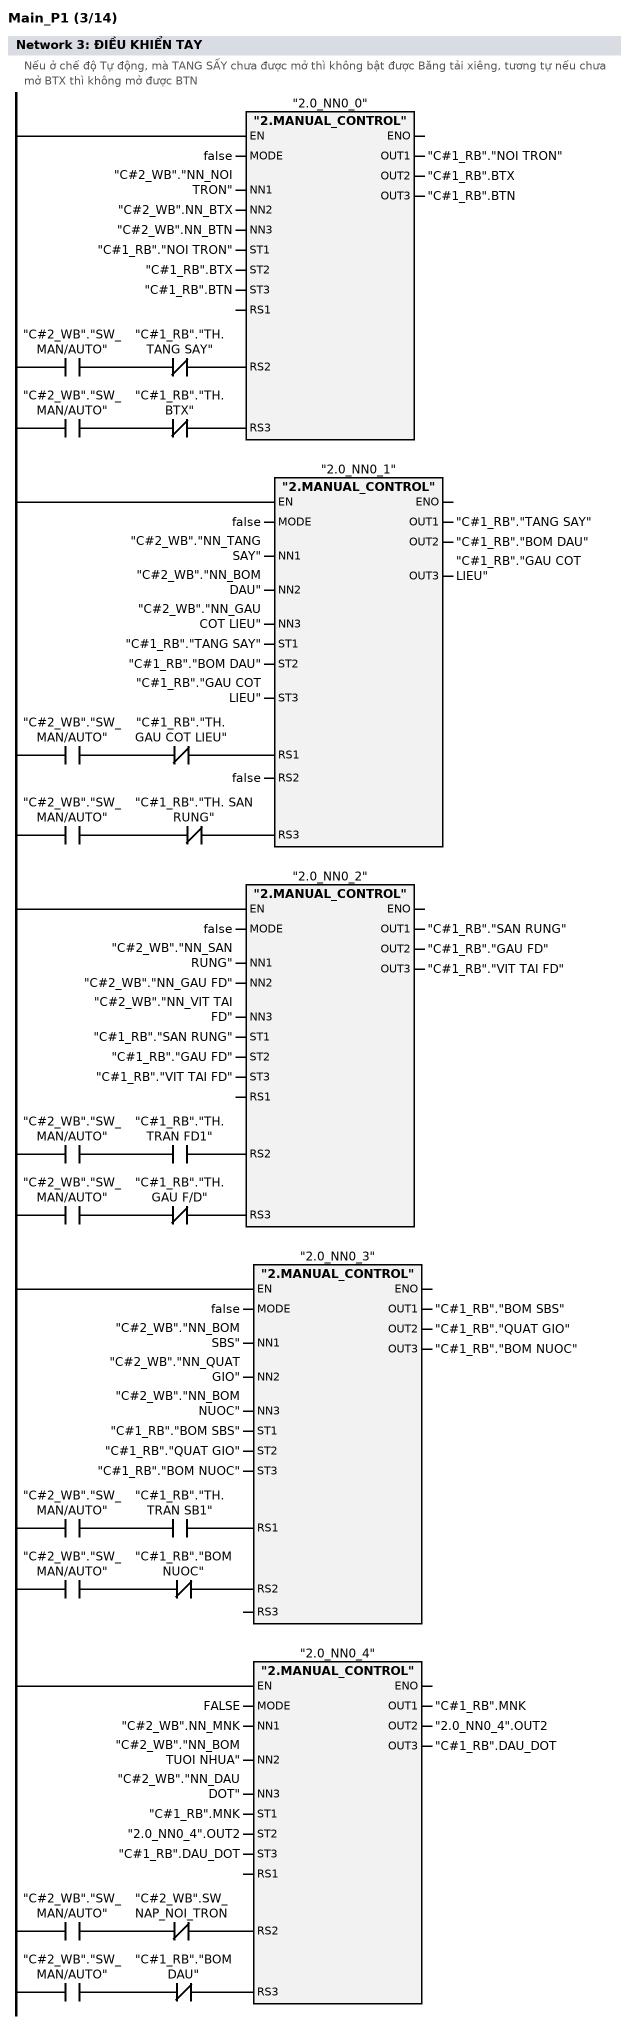
   RUNG wire#powerrail
      "2.0_NN0_0"(RS2 := wire#w1, RS3 := wire#w2, MODE := false, NN1 := "C#2_WB"."NN_NOI TRON", NN2 := "C#2_WB".NN_BTX, NN3 := "C#2_WB".NN_BTN, ST1 := "C#1_RB"."NOI TRON", ST2 := "C#1_RB".BTX, ST3 := "C#1_RB".BTN, RS1 :=, OUT1 => "C#1_RB"."NOI TRON", OUT2 => "C#1_RB".BTX, OUT3 => "C#1_RB".BTN)
   END_RUNG
   RUNG wire#powerrail
      Contact( "C#2_WB"."SW_MAN/AUTO" )
      I_Contact( "C#1_RB"."TH. TANG SAY" )
   END_RUNG wire#w1
   RUNG wire#powerrail
      Contact( "C#2_WB"."SW_MAN/AUTO" )
      I_Contact( "C#1_RB"."TH. BTX" )
   END_RUNG wire#w2
   RUNG wire#powerrail
      "2.0_NN0_1"(RS1 := wire#w3, RS3 := wire#w4, MODE := false, NN1 := "C#2_WB"."NN_TANG SAY", NN2 := "C#2_WB"."NN_BOM DAU", NN3 := "C#2_WB"."NN_GAU COT LIEU", ST1 := "C#1_RB"."TANG SAY", ST2 := "C#1_RB"."BOM DAU", ST3 := "C#1_RB"."GAU COT LIEU", RS2 := false, OUT1 => "C#1_RB"."TANG SAY", OUT2 => "C#1_RB"."BOM DAU", OUT3 => "C#1_RB"."GAU COT LIEU")
   END_RUNG
   RUNG wire#powerrail
      Contact( "C#2_WB"."SW_MAN/AUTO" )
      I_Contact( "C#1_RB"."TH. GAU COT LIEU" )
   END_RUNG wire#w3
   RUNG wire#powerrail
      Contact( "C#2_WB"."SW_MAN/AUTO" )
      I_Contact( "C#1_RB"."TH. SAN RUNG" )
   END_RUNG wire#w4
   RUNG wire#powerrail
      "2.0_NN0_2"(RS2 := wire#w5, RS3 := wire#w6, MODE := false, NN1 := "C#2_WB"."NN_SAN RUNG", NN2 := "C#2_WB"."NN_GAU FD", NN3 := "C#2_WB"."NN_VIT TAI FD", ST1 := "C#1_RB"."SAN RUNG", ST2 := "C#1_RB"."GAU FD", ST3 := "C#1_RB"."VIT TAI FD", RS1 :=, OUT1 => "C#1_RB"."SAN RUNG", OUT2 => "C#1_RB"."GAU FD", OUT3 => "C#1_RB"."VIT TAI FD")
   END_RUNG
   RUNG wire#powerrail
      Contact( "C#2_WB"."SW_MAN/AUTO" )
      Contact( "C#1_RB"."TH. TRAN FD1" )
   END_RUNG wire#w5
   RUNG wire#powerrail
      Contact( "C#2_WB"."SW_MAN/AUTO" )
      I_Contact( "C#1_RB"."TH. GAU F/D" )
   END_RUNG wire#w6
   RUNG wire#powerrail
      "2.0_NN0_3"(RS1 := wire#w7, RS2 := wire#w8, MODE := false, NN1 := "C#2_WB"."NN_BOM SBS", NN2 := "C#2_WB"."NN_QUAT GIO", NN3 := "C#2_WB"."NN_BOM NUOC", ST1 := "C#1_RB"."BOM SBS", ST2 := "C#1_RB"."QUAT GIO", ST3 := "C#1_RB"."BOM NUOC", RS3 :=, OUT1 => "C#1_RB"."BOM SBS", OUT2 => "C#1_RB"."QUAT GIO", OUT3 => "C#1_RB"."BOM NUOC")
   END_RUNG
   RUNG wire#powerrail
      Contact( "C#2_WB"."SW_MAN/AUTO" )
      Contact( "C#1_RB"."TH. TRAN SB1" )
   END_RUNG wire#w7
   RUNG wire#powerrail
      Contact( "C#2_WB"."SW_MAN/AUTO" )
      I_Contact( "C#1_RB"."BOM NUOC" )
   END_RUNG wire#w8
   RUNG wire#powerrail
      "2.0_NN0_4"(RS2 := wire#w9, RS3 := wire#w10, MODE := FALSE, NN1 := "C#2_WB".NN_MNK, NN2 := "C#2_WB"."NN_BOM TUOI NHUA", NN3 := "C#2_WB"."NN_DAU DOT", ST1 := "C#1_RB".MNK, ST2 := "2.0_NN0_4".OUT2, ST3 := "C#1_RB".DAU_DOT, RS1 :=, OUT1 => "C#1_RB".MNK, OUT2 => "2.0_NN0_4".OUT2, OUT3 => "C#1_RB".DAU_DOT)
   END_RUNG
   RUNG wire#powerrail
      Contact( "C#2_WB"."SW_MAN/AUTO" )
      I_Contact( "C#2_WB".SW_NAP_NOI_TRON )
   END_RUNG wire#w9
   RUNG wire#powerrail
      Contact( "C#2_WB"."SW_MAN/AUTO" )
      I_Contact( "C#1_RB"."BOM DAU" )
   END_RUNG wire#w10
   // the same network as SCL:
   "2.0_NN0_0"(MODE := false,   // "2.MANUAL_CONTROL"
               NN1 := "C#2_WB"."NN_NOI TRON",
               NN2 := "C#2_WB".NN_BTX,
               NN3 := "C#2_WB".NN_BTN,
               ST1 := "C#1_RB"."NOI TRON",
               ST2 := "C#1_RB".BTX,
               ST3 := "C#1_RB".BTN,
               RS2 := "C#2_WB"."SW_MAN/AUTO" AND NOT "C#1_RB"."TH. TANG SAY",
               RS3 := "C#2_WB"."SW_MAN/AUTO" AND NOT "C#1_RB"."TH. BTX",
               OUT1 => "C#1_RB"."NOI TRON",
               OUT2 => "C#1_RB".BTX,
               OUT3 => "C#1_RB".BTN);
   "2.0_NN0_1"(MODE := false,   // "2.MANUAL_CONTROL"
               NN1 := "C#2_WB"."NN_TANG SAY",
               NN2 := "C#2_WB"."NN_BOM DAU",
               NN3 := "C#2_WB"."NN_GAU COT LIEU",
               ST1 := "C#1_RB"."TANG SAY",
               ST2 := "C#1_RB"."BOM DAU",
               ST3 := "C#1_RB"."GAU COT LIEU",
               RS1 := "C#2_WB"."SW_MAN/AUTO" AND NOT "C#1_RB"."TH. GAU COT LIEU",
               RS2 := false,
               RS3 := "C#2_WB"."SW_MAN/AUTO" AND NOT "C#1_RB"."TH. SAN RUNG",
               OUT1 => "C#1_RB"."TANG SAY",
               OUT2 => "C#1_RB"."BOM DAU",
               OUT3 => "C#1_RB"."GAU COT LIEU");
   "2.0_NN0_2"(MODE := false,   // "2.MANUAL_CONTROL"
               NN1 := "C#2_WB"."NN_SAN RUNG",
               NN2 := "C#2_WB"."NN_GAU FD",
               NN3 := "C#2_WB"."NN_VIT TAI FD",
               ST1 := "C#1_RB"."SAN RUNG",
               ST2 := "C#1_RB"."GAU FD",
               ST3 := "C#1_RB"."VIT TAI FD",
               RS2 := "C#2_WB"."SW_MAN/AUTO" AND "C#1_RB"."TH. TRAN FD1",
               RS3 := "C#2_WB"."SW_MAN/AUTO" AND NOT "C#1_RB"."TH. GAU F/D",
               OUT1 => "C#1_RB"."SAN RUNG",
               OUT2 => "C#1_RB"."GAU FD",
               OUT3 => "C#1_RB"."VIT TAI FD");
   "2.0_NN0_3"(MODE := false,   // "2.MANUAL_CONTROL"
               NN1 := "C#2_WB"."NN_BOM SBS",
               NN2 := "C#2_WB"."NN_QUAT GIO",
               NN3 := "C#2_WB"."NN_BOM NUOC",
               ST1 := "C#1_RB"."BOM SBS",
               ST2 := "C#1_RB"."QUAT GIO",
               ST3 := "C#1_RB"."BOM NUOC",
               RS1 := "C#2_WB"."SW_MAN/AUTO" AND "C#1_RB"."TH. TRAN SB1",
               RS2 := "C#2_WB"."SW_MAN/AUTO" AND NOT "C#1_RB"."BOM NUOC",
               OUT1 => "C#1_RB"."BOM SBS",
               OUT2 => "C#1_RB"."QUAT GIO",
               OUT3 => "C#1_RB"."BOM NUOC");
   "2.0_NN0_4"(MODE := FALSE,   // "2.MANUAL_CONTROL"
               NN1 := "C#2_WB".NN_MNK,
               NN2 := "C#2_WB"."NN_BOM TUOI NHUA",
               NN3 := "C#2_WB"."NN_DAU DOT",
               ST1 := "C#1_RB".MNK,
               ST2 := "2.0_NN0_4".OUT2,
               ST3 := "C#1_RB".DAU_DOT,
               RS2 := "C#2_WB"."SW_MAN/AUTO" AND NOT "C#2_WB".SW_NAP_NOI_TRON,
               RS3 := "C#2_WB"."SW_MAN/AUTO" AND NOT "C#1_RB"."BOM DAU",
               OUT1 => "C#1_RB".MNK,
               OUT2 => "2.0_NN0_4".OUT2,
               OUT3 => "C#1_RB".DAU_DOT);
END_REGION

REGION Network 4: CONVERT ANALOG IN PUT (0.0/ 0-10V: 1.0/4-20mA: 2.0/0-20mA)
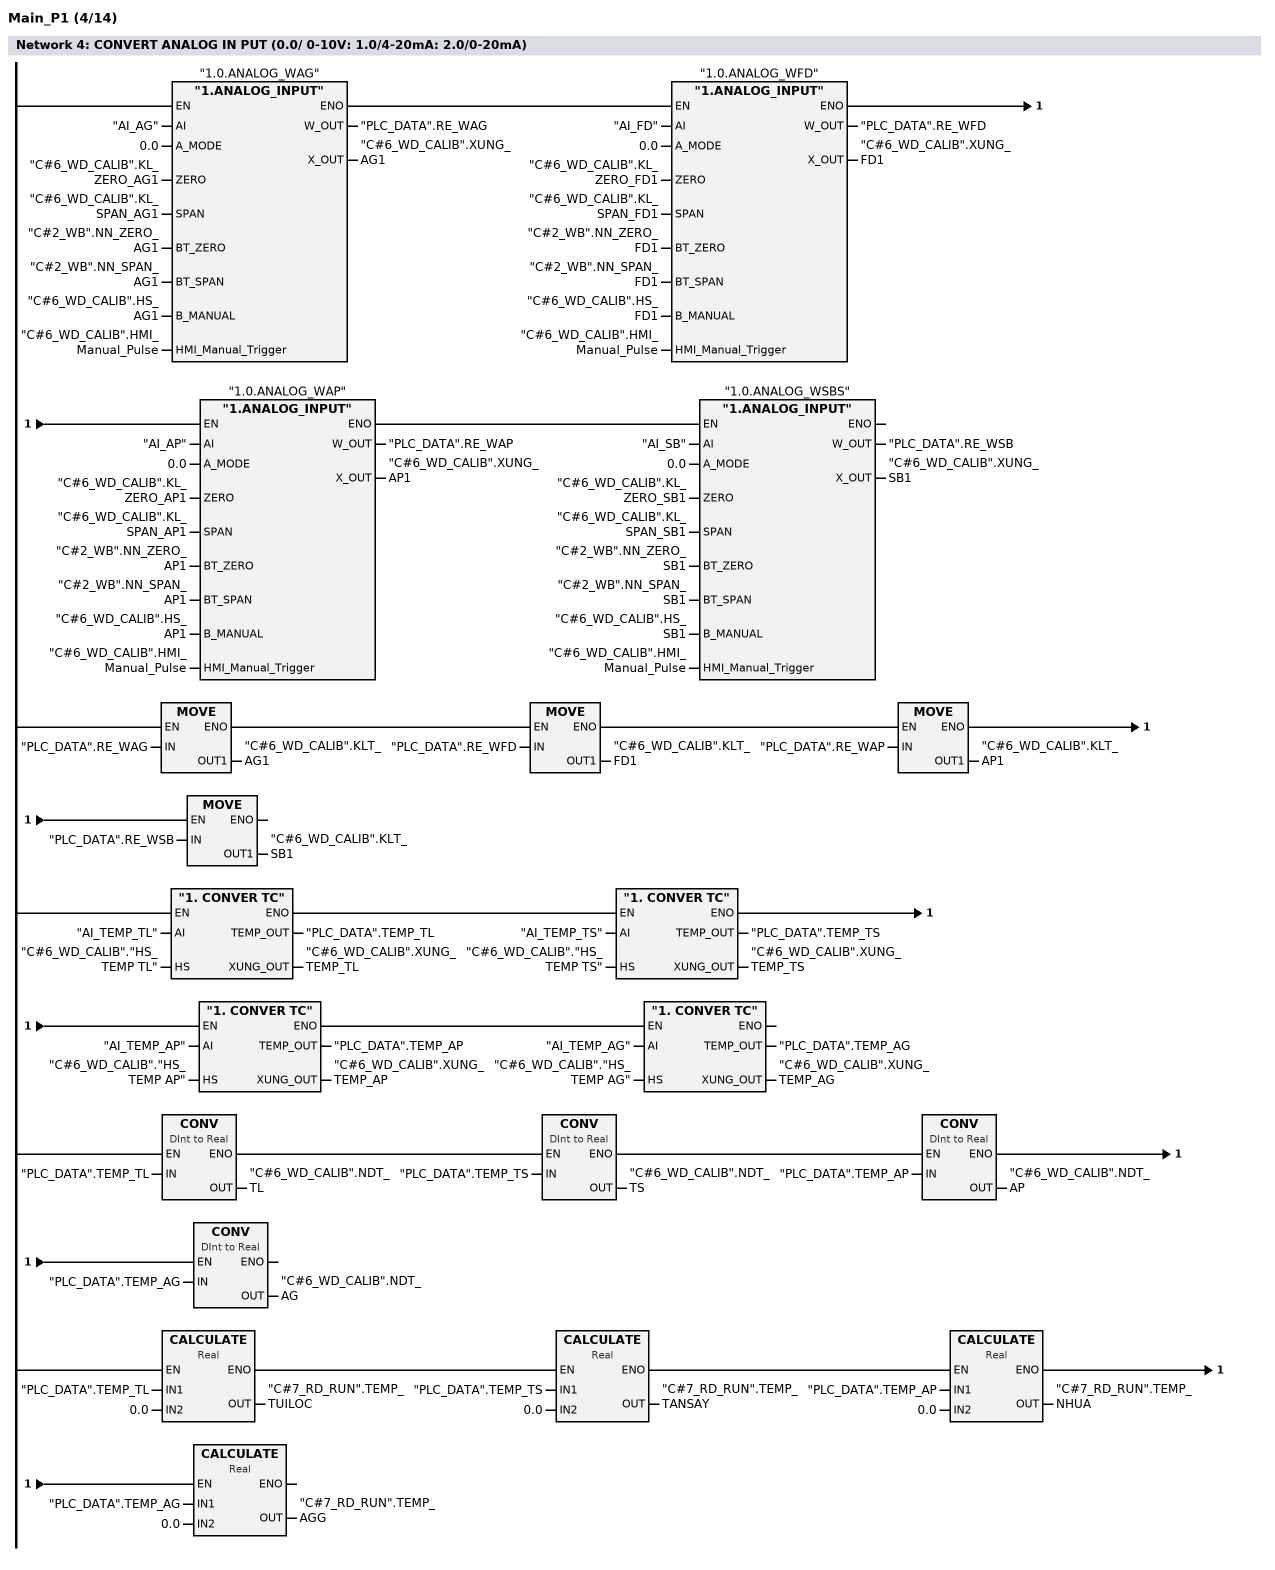
   RUNG wire#powerrail
      "1.0.ANALOG_WAG"(AI := "AI_AG", A_MODE := 0.0, ZERO := "C#6_WD_CALIB".KL_ZERO_AG1, SPAN := "C#6_WD_CALIB".KL_SPAN_AG1, BT_ZERO := "C#2_WB".NN_ZERO_AG1, BT_SPAN := "C#2_WB".NN_SPAN_AG1, B_MANUAL := "C#6_WD_CALIB".HS_AG1, HMI_Manual_Trigger := "C#6_WD_CALIB".HMI_Manual_Pulse, W_OUT => "PLC_DATA".RE_WAG, X_OUT => "C#6_WD_CALIB".XUNG_AG1)
      "1.0.ANALOG_WFD"(AI := "AI_FD", A_MODE := 0.0, ZERO := "C#6_WD_CALIB".KL_ZERO_FD1, SPAN := "C#6_WD_CALIB".KL_SPAN_FD1, BT_ZERO := "C#2_WB".NN_ZERO_FD1, BT_SPAN := "C#2_WB".NN_SPAN_FD1, B_MANUAL := "C#6_WD_CALIB".HS_FD1, HMI_Manual_Trigger := "C#6_WD_CALIB".HMI_Manual_Pulse, W_OUT => "PLC_DATA".RE_WFD, X_OUT => "C#6_WD_CALIB".XUNG_FD1)
      "1.0.ANALOG_WAP"(AI := "AI_AP", A_MODE := 0.0, ZERO := "C#6_WD_CALIB".KL_ZERO_AP1, SPAN := "C#6_WD_CALIB".KL_SPAN_AP1, BT_ZERO := "C#2_WB".NN_ZERO_AP1, BT_SPAN := "C#2_WB".NN_SPAN_AP1, B_MANUAL := "C#6_WD_CALIB".HS_AP1, HMI_Manual_Trigger := "C#6_WD_CALIB".HMI_Manual_Pulse, W_OUT => "PLC_DATA".RE_WAP, X_OUT => "C#6_WD_CALIB".XUNG_AP1)
      "1.0.ANALOG_WSBS"(AI := "AI_SB", A_MODE := 0.0, ZERO := "C#6_WD_CALIB".KL_ZERO_SB1, SPAN := "C#6_WD_CALIB".KL_SPAN_SB1, BT_ZERO := "C#2_WB".NN_ZERO_SB1, BT_SPAN := "C#2_WB".NN_SPAN_SB1, B_MANUAL := "C#6_WD_CALIB".HS_SB1, HMI_Manual_Trigger := "C#6_WD_CALIB".HMI_Manual_Pulse, W_OUT => "PLC_DATA".RE_WSB, X_OUT => "C#6_WD_CALIB".XUNG_SB1)
   END_RUNG
   RUNG wire#powerrail
      { S7_GenerateENO := "TRUE" } Move(in := "PLC_DATA".RE_WAG, out1 => "C#6_WD_CALIB".KLT_AG1)
      { S7_GenerateENO := "TRUE" } Move(in := "PLC_DATA".RE_WFD, out1 => "C#6_WD_CALIB".KLT_FD1)
      { S7_GenerateENO := "TRUE" } Move(in := "PLC_DATA".RE_WAP, out1 => "C#6_WD_CALIB".KLT_AP1)
      { S7_GenerateENO := "TRUE" } Move(in := "PLC_DATA".RE_WSB, out1 => "C#6_WD_CALIB".KLT_SB1)
   END_RUNG
   RUNG wire#powerrail
      "1. CONVER TC"(AI := "AI_TEMP_TL", HS := "C#6_WD_CALIB"."HS_TEMP TL", TEMP_OUT => "PLC_DATA".TEMP_TL, XUNG_OUT => "C#6_WD_CALIB".XUNG_TEMP_TL)
      "1. CONVER TC"(AI := "AI_TEMP_TS", HS := "C#6_WD_CALIB"."HS_TEMP TS", TEMP_OUT => "PLC_DATA".TEMP_TS, XUNG_OUT => "C#6_WD_CALIB".XUNG_TEMP_TS)
      "1. CONVER TC"(AI := "AI_TEMP_AP", HS := "C#6_WD_CALIB"."HS_TEMP AP", TEMP_OUT => "PLC_DATA".TEMP_AP, XUNG_OUT => "C#6_WD_CALIB".XUNG_TEMP_AP)
      "1. CONVER TC"(AI := "AI_TEMP_AG", HS := "C#6_WD_CALIB"."HS_TEMP AG", TEMP_OUT => "PLC_DATA".TEMP_AG, XUNG_OUT => "C#6_WD_CALIB".XUNG_TEMP_AG)
   END_RUNG
   RUNG wire#powerrail
      { S7_Templates := "[SrcType := DInt, DestType := Real]" } Convert(in := "PLC_DATA".TEMP_TL, out => "C#6_WD_CALIB".NDT_TL)
      { S7_Templates := "[SrcType := DInt, DestType := Real]" } Convert(in := "PLC_DATA".TEMP_TS, out => "C#6_WD_CALIB".NDT_TS)
      { S7_Templates := "[SrcType := DInt, DestType := Real]" } Convert(in := "PLC_DATA".TEMP_AP, out => "C#6_WD_CALIB".NDT_AP)
      { S7_Templates := "[SrcType := DInt, DestType := Real]" } Convert(in := "PLC_DATA".TEMP_AG, out => "C#6_WD_CALIB".NDT_AG)
   END_RUNG
   RUNG wire#powerrail
      { S7_Templates := "SrcType := Real"; S7_Expression := "IN1+IN2" } Calculate(in1 := "PLC_DATA".TEMP_TL, in2 := 0.0, out => "C#7_RD_RUN".TEMP_TUILOC)
      { S7_Templates := "SrcType := Real"; S7_Expression := "IN1+IN2" } Calculate(in1 := "PLC_DATA".TEMP_TS, in2 := 0.0, out => "C#7_RD_RUN".TEMP_TANSAY)
      { S7_Templates := "SrcType := Real"; S7_Expression := "IN1+IN2" } Calculate(in1 := "PLC_DATA".TEMP_AP, in2 := 0.0, out => "C#7_RD_RUN".TEMP_NHUA)
      { S7_Templates := "SrcType := Real"; S7_Expression := "IN1+IN2" } Calculate(in1 := "PLC_DATA".TEMP_AG, in2 := 0.0, out => "C#7_RD_RUN".TEMP_AGG)
   END_RUNG
   // the same network as SCL:
   // ENO of a box is taken as its EN; it also drops when the box reports an error
   "1.0.ANALOG_WAG"(AI := "AI_AG",   // "1.ANALOG_INPUT"
                    A_MODE := 0.0,
                    ZERO := "C#6_WD_CALIB".KL_ZERO_AG1,
                    SPAN := "C#6_WD_CALIB".KL_SPAN_AG1,
                    BT_ZERO := "C#2_WB".NN_ZERO_AG1,
                    BT_SPAN := "C#2_WB".NN_SPAN_AG1,
                    B_MANUAL := "C#6_WD_CALIB".HS_AG1,
                    HMI_Manual_Trigger := "C#6_WD_CALIB".HMI_Manual_Pulse,
                    W_OUT => "PLC_DATA".RE_WAG,
                    X_OUT => "C#6_WD_CALIB".XUNG_AG1,
                    ENO => #_w1);
   "1.0.ANALOG_WFD"(EN := #_w1,   // "1.ANALOG_INPUT"
                    AI := "AI_FD",
                    A_MODE := 0.0,
                    ZERO := "C#6_WD_CALIB".KL_ZERO_FD1,
                    SPAN := "C#6_WD_CALIB".KL_SPAN_FD1,
                    BT_ZERO := "C#2_WB".NN_ZERO_FD1,
                    BT_SPAN := "C#2_WB".NN_SPAN_FD1,
                    B_MANUAL := "C#6_WD_CALIB".HS_FD1,
                    HMI_Manual_Trigger := "C#6_WD_CALIB".HMI_Manual_Pulse,
                    W_OUT => "PLC_DATA".RE_WFD,
                    X_OUT => "C#6_WD_CALIB".XUNG_FD1,
                    ENO => #_w2);
   "1.0.ANALOG_WAP"(EN := #_w2,   // "1.ANALOG_INPUT"
                    AI := "AI_AP",
                    A_MODE := 0.0,
                    ZERO := "C#6_WD_CALIB".KL_ZERO_AP1,
                    SPAN := "C#6_WD_CALIB".KL_SPAN_AP1,
                    BT_ZERO := "C#2_WB".NN_ZERO_AP1,
                    BT_SPAN := "C#2_WB".NN_SPAN_AP1,
                    B_MANUAL := "C#6_WD_CALIB".HS_AP1,
                    HMI_Manual_Trigger := "C#6_WD_CALIB".HMI_Manual_Pulse,
                    W_OUT => "PLC_DATA".RE_WAP,
                    X_OUT => "C#6_WD_CALIB".XUNG_AP1,
                    ENO => #_w3);
   IF #_w3 THEN
       "1.0.ANALOG_WSBS"(AI := "AI_SB",   // "1.ANALOG_INPUT"
                         A_MODE := 0.0,
                         ZERO := "C#6_WD_CALIB".KL_ZERO_SB1,
                         SPAN := "C#6_WD_CALIB".KL_SPAN_SB1,
                         BT_ZERO := "C#2_WB".NN_ZERO_SB1,
                         BT_SPAN := "C#2_WB".NN_SPAN_SB1,
                         B_MANUAL := "C#6_WD_CALIB".HS_SB1,
                         HMI_Manual_Trigger := "C#6_WD_CALIB".HMI_Manual_Pulse,
                         W_OUT => "PLC_DATA".RE_WSB,
                         X_OUT => "C#6_WD_CALIB".XUNG_SB1);
   END_IF;
   "C#6_WD_CALIB".KLT_AG1 := "PLC_DATA".RE_WAG;
   "C#6_WD_CALIB".KLT_FD1 := "PLC_DATA".RE_WFD;
   "C#6_WD_CALIB".KLT_AP1 := "PLC_DATA".RE_WAP;
   "C#6_WD_CALIB".KLT_SB1 := "PLC_DATA".RE_WSB;
   "1. CONVER TC"(AI := "AI_TEMP_TL",
                  HS := "C#6_WD_CALIB"."HS_TEMP TL",
                  TEMP_OUT => "PLC_DATA".TEMP_TL,
                  XUNG_OUT => "C#6_WD_CALIB".XUNG_TEMP_TL,
                  ENO => #_w4);
   "1. CONVER TC"(EN := #_w4,
                  AI := "AI_TEMP_TS",
                  HS := "C#6_WD_CALIB"."HS_TEMP TS",
                  TEMP_OUT => "PLC_DATA".TEMP_TS,
                  XUNG_OUT => "C#6_WD_CALIB".XUNG_TEMP_TS,
                  ENO => #_w5);
   "1. CONVER TC"(EN := #_w5,
                  AI := "AI_TEMP_AP",
                  HS := "C#6_WD_CALIB"."HS_TEMP AP",
                  TEMP_OUT => "PLC_DATA".TEMP_AP,
                  XUNG_OUT => "C#6_WD_CALIB".XUNG_TEMP_AP,
                  ENO => #_w6);
   IF #_w6 THEN
       "1. CONVER TC"(AI := "AI_TEMP_AG",
                      HS := "C#6_WD_CALIB"."HS_TEMP AG",
                      TEMP_OUT => "PLC_DATA".TEMP_AG,
                      XUNG_OUT => "C#6_WD_CALIB".XUNG_TEMP_AG);
   END_IF;
   "C#6_WD_CALIB".NDT_TL := DINT_TO_REAL("PLC_DATA".TEMP_TL);
   "C#6_WD_CALIB".NDT_TS := DINT_TO_REAL("PLC_DATA".TEMP_TS);
   "C#6_WD_CALIB".NDT_AP := DINT_TO_REAL("PLC_DATA".TEMP_AP);
   "C#6_WD_CALIB".NDT_AG := DINT_TO_REAL("PLC_DATA".TEMP_AG);
   "C#7_RD_RUN".TEMP_TUILOC := "PLC_DATA".TEMP_TL+0.0;
   "C#7_RD_RUN".TEMP_TANSAY := "PLC_DATA".TEMP_TS+0.0;
   "C#7_RD_RUN".TEMP_NHUA := "PLC_DATA".TEMP_AP+0.0;
   "C#7_RD_RUN".TEMP_AGG := "PLC_DATA".TEMP_AG+0.0;
END_REGION

REGION Network 5: CONVERT ANALOG IN PUT (0.0/ 0-10V: 1.0/4-20mA: 2.0/0-20mA) - Mode Độc Lập
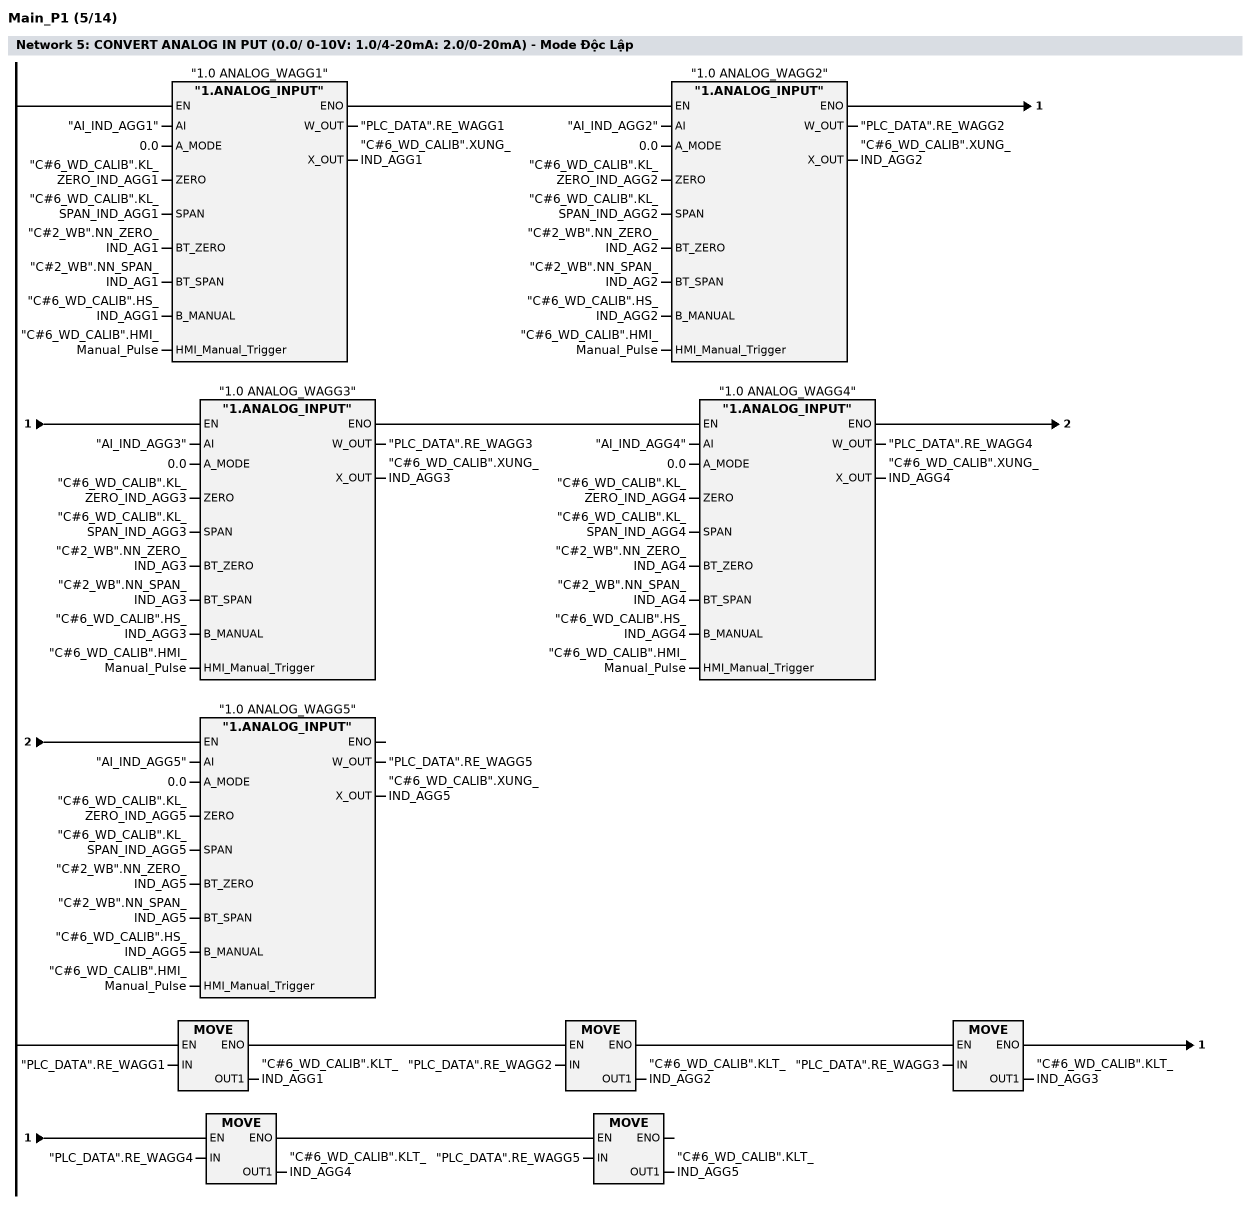
   RUNG wire#powerrail
      "1.0 ANALOG_WAGG1"(AI := "AI_IND_AGG1", A_MODE := 0.0, ZERO := "C#6_WD_CALIB".KL_ZERO_IND_AGG1, SPAN := "C#6_WD_CALIB".KL_SPAN_IND_AGG1, BT_ZERO := "C#2_WB".NN_ZERO_IND_AG1, BT_SPAN := "C#2_WB".NN_SPAN_IND_AG1, B_MANUAL := "C#6_WD_CALIB".HS_IND_AGG1, HMI_Manual_Trigger := "C#6_WD_CALIB".HMI_Manual_Pulse, W_OUT => "PLC_DATA".RE_WAGG1, X_OUT => "C#6_WD_CALIB".XUNG_IND_AGG1)
      "1.0 ANALOG_WAGG2"(AI := "AI_IND_AGG2", A_MODE := 0.0, ZERO := "C#6_WD_CALIB".KL_ZERO_IND_AGG2, SPAN := "C#6_WD_CALIB".KL_SPAN_IND_AGG2, BT_ZERO := "C#2_WB".NN_ZERO_IND_AG2, BT_SPAN := "C#2_WB".NN_SPAN_IND_AG2, B_MANUAL := "C#6_WD_CALIB".HS_IND_AGG2, HMI_Manual_Trigger := "C#6_WD_CALIB".HMI_Manual_Pulse, W_OUT => "PLC_DATA".RE_WAGG2, X_OUT => "C#6_WD_CALIB".XUNG_IND_AGG2)
      "1.0 ANALOG_WAGG3"(AI := "AI_IND_AGG3", A_MODE := 0.0, ZERO := "C#6_WD_CALIB".KL_ZERO_IND_AGG3, SPAN := "C#6_WD_CALIB".KL_SPAN_IND_AGG3, BT_ZERO := "C#2_WB".NN_ZERO_IND_AG3, BT_SPAN := "C#2_WB".NN_SPAN_IND_AG3, B_MANUAL := "C#6_WD_CALIB".HS_IND_AGG3, HMI_Manual_Trigger := "C#6_WD_CALIB".HMI_Manual_Pulse, W_OUT => "PLC_DATA".RE_WAGG3, X_OUT => "C#6_WD_CALIB".XUNG_IND_AGG3)
      "1.0 ANALOG_WAGG4"(AI := "AI_IND_AGG4", A_MODE := 0.0, ZERO := "C#6_WD_CALIB".KL_ZERO_IND_AGG4, SPAN := "C#6_WD_CALIB".KL_SPAN_IND_AGG4, BT_ZERO := "C#2_WB".NN_ZERO_IND_AG4, BT_SPAN := "C#2_WB".NN_SPAN_IND_AG4, B_MANUAL := "C#6_WD_CALIB".HS_IND_AGG4, HMI_Manual_Trigger := "C#6_WD_CALIB".HMI_Manual_Pulse, W_OUT => "PLC_DATA".RE_WAGG4, X_OUT => "C#6_WD_CALIB".XUNG_IND_AGG4)
      "1.0 ANALOG_WAGG5"(AI := "AI_IND_AGG5", A_MODE := 0.0, ZERO := "C#6_WD_CALIB".KL_ZERO_IND_AGG5, SPAN := "C#6_WD_CALIB".KL_SPAN_IND_AGG5, BT_ZERO := "C#2_WB".NN_ZERO_IND_AG5, BT_SPAN := "C#2_WB".NN_SPAN_IND_AG5, B_MANUAL := "C#6_WD_CALIB".HS_IND_AGG5, HMI_Manual_Trigger := "C#6_WD_CALIB".HMI_Manual_Pulse, W_OUT => "PLC_DATA".RE_WAGG5, X_OUT => "C#6_WD_CALIB".XUNG_IND_AGG5)
   END_RUNG
   RUNG wire#powerrail
      { S7_GenerateENO := "TRUE" } Move(in := "PLC_DATA".RE_WAGG1, out1 => "C#6_WD_CALIB".KLT_IND_AGG1)
      { S7_GenerateENO := "TRUE" } Move(in := "PLC_DATA".RE_WAGG2, out1 => "C#6_WD_CALIB".KLT_IND_AGG2)
      { S7_GenerateENO := "TRUE" } Move(in := "PLC_DATA".RE_WAGG3, out1 => "C#6_WD_CALIB".KLT_IND_AGG3)
      { S7_GenerateENO := "TRUE" } Move(in := "PLC_DATA".RE_WAGG4, out1 => "C#6_WD_CALIB".KLT_IND_AGG4)
      { S7_GenerateENO := "TRUE" } Move(in := "PLC_DATA".RE_WAGG5, out1 => "C#6_WD_CALIB".KLT_IND_AGG5)
   END_RUNG
   // the same network as SCL:
   // ENO of a box is taken as its EN; it also drops when the box reports an error
   "1.0 ANALOG_WAGG1"(AI := "AI_IND_AGG1",   // "1.ANALOG_INPUT"
                      A_MODE := 0.0,
                      ZERO := "C#6_WD_CALIB".KL_ZERO_IND_AGG1,
                      SPAN := "C#6_WD_CALIB".KL_SPAN_IND_AGG1,
                      BT_ZERO := "C#2_WB".NN_ZERO_IND_AG1,
                      BT_SPAN := "C#2_WB".NN_SPAN_IND_AG1,
                      B_MANUAL := "C#6_WD_CALIB".HS_IND_AGG1,
                      HMI_Manual_Trigger := "C#6_WD_CALIB".HMI_Manual_Pulse,
                      W_OUT => "PLC_DATA".RE_WAGG1,
                      X_OUT => "C#6_WD_CALIB".XUNG_IND_AGG1,
                      ENO => #_w1);
   "1.0 ANALOG_WAGG2"(EN := #_w1,   // "1.ANALOG_INPUT"
                      AI := "AI_IND_AGG2",
                      A_MODE := 0.0,
                      ZERO := "C#6_WD_CALIB".KL_ZERO_IND_AGG2,
                      SPAN := "C#6_WD_CALIB".KL_SPAN_IND_AGG2,
                      BT_ZERO := "C#2_WB".NN_ZERO_IND_AG2,
                      BT_SPAN := "C#2_WB".NN_SPAN_IND_AG2,
                      B_MANUAL := "C#6_WD_CALIB".HS_IND_AGG2,
                      HMI_Manual_Trigger := "C#6_WD_CALIB".HMI_Manual_Pulse,
                      W_OUT => "PLC_DATA".RE_WAGG2,
                      X_OUT => "C#6_WD_CALIB".XUNG_IND_AGG2,
                      ENO => #_w2);
   "1.0 ANALOG_WAGG3"(EN := #_w2,   // "1.ANALOG_INPUT"
                      AI := "AI_IND_AGG3",
                      A_MODE := 0.0,
                      ZERO := "C#6_WD_CALIB".KL_ZERO_IND_AGG3,
                      SPAN := "C#6_WD_CALIB".KL_SPAN_IND_AGG3,
                      BT_ZERO := "C#2_WB".NN_ZERO_IND_AG3,
                      BT_SPAN := "C#2_WB".NN_SPAN_IND_AG3,
                      B_MANUAL := "C#6_WD_CALIB".HS_IND_AGG3,
                      HMI_Manual_Trigger := "C#6_WD_CALIB".HMI_Manual_Pulse,
                      W_OUT => "PLC_DATA".RE_WAGG3,
                      X_OUT => "C#6_WD_CALIB".XUNG_IND_AGG3,
                      ENO => #_w3);
   "1.0 ANALOG_WAGG4"(EN := #_w3,   // "1.ANALOG_INPUT"
                      AI := "AI_IND_AGG4",
                      A_MODE := 0.0,
                      ZERO := "C#6_WD_CALIB".KL_ZERO_IND_AGG4,
                      SPAN := "C#6_WD_CALIB".KL_SPAN_IND_AGG4,
                      BT_ZERO := "C#2_WB".NN_ZERO_IND_AG4,
                      BT_SPAN := "C#2_WB".NN_SPAN_IND_AG4,
                      B_MANUAL := "C#6_WD_CALIB".HS_IND_AGG4,
                      HMI_Manual_Trigger := "C#6_WD_CALIB".HMI_Manual_Pulse,
                      W_OUT => "PLC_DATA".RE_WAGG4,
                      X_OUT => "C#6_WD_CALIB".XUNG_IND_AGG4,
                      ENO => #_w4);
   IF #_w4 THEN
       "1.0 ANALOG_WAGG5"(AI := "AI_IND_AGG5",   // "1.ANALOG_INPUT"
                          A_MODE := 0.0,
                          ZERO := "C#6_WD_CALIB".KL_ZERO_IND_AGG5,
                          SPAN := "C#6_WD_CALIB".KL_SPAN_IND_AGG5,
                          BT_ZERO := "C#2_WB".NN_ZERO_IND_AG5,
                          BT_SPAN := "C#2_WB".NN_SPAN_IND_AG5,
                          B_MANUAL := "C#6_WD_CALIB".HS_IND_AGG5,
                          HMI_Manual_Trigger := "C#6_WD_CALIB".HMI_Manual_Pulse,
                          W_OUT => "PLC_DATA".RE_WAGG5,
                          X_OUT => "C#6_WD_CALIB".XUNG_IND_AGG5);
   END_IF;
   "C#6_WD_CALIB".KLT_IND_AGG1 := "PLC_DATA".RE_WAGG1;
   "C#6_WD_CALIB".KLT_IND_AGG2 := "PLC_DATA".RE_WAGG2;
   "C#6_WD_CALIB".KLT_IND_AGG3 := "PLC_DATA".RE_WAGG3;
   "C#6_WD_CALIB".KLT_IND_AGG4 := "PLC_DATA".RE_WAGG4;
   "C#6_WD_CALIB".KLT_IND_AGG5 := "PLC_DATA".RE_WAGG5;
END_REGION

REGION Network 6: RUN MODE
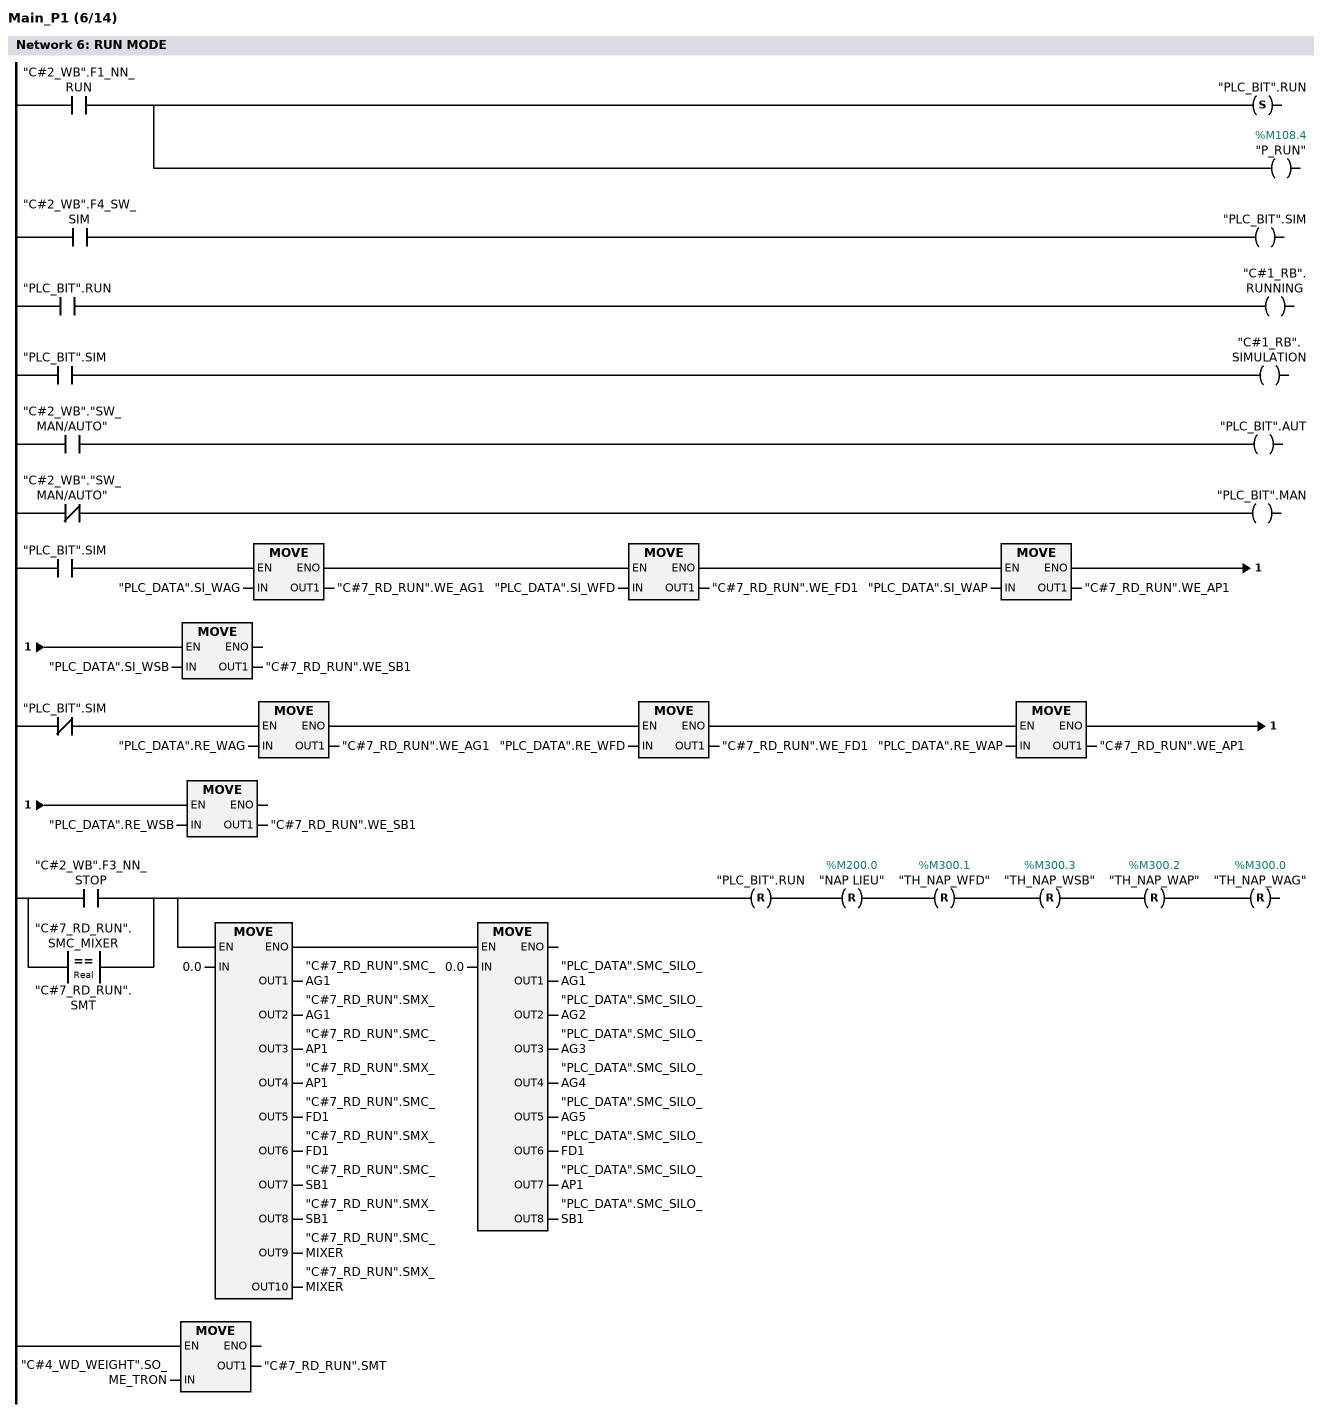
   RUNG wire#powerrail
      Contact( "C#2_WB".F1_NN_RUN )
      wire#w1
      S_Coil( "PLC_BIT".RUN )
   END_RUNG
   RUNG wire#w1
      Coil( "P_RUN" )
   END_RUNG
   RUNG wire#powerrail
      Contact( "C#2_WB".F4_SW_SIM )
      Coil( "PLC_BIT".SIM )
   END_RUNG
   RUNG wire#powerrail
      Contact( "PLC_BIT".RUN )
      Coil( "C#1_RB".RUNNING )
   END_RUNG
   RUNG wire#powerrail
      Contact( "PLC_BIT".SIM )
      Coil( "C#1_RB".SIMULATION )
   END_RUNG
   RUNG wire#powerrail
      Contact( "C#2_WB"."SW_MAN/AUTO" )
      Coil( "PLC_BIT".AUT )
   END_RUNG
   RUNG wire#powerrail
      I_Contact( "C#2_WB"."SW_MAN/AUTO" )
      Coil( "PLC_BIT".MAN )
   END_RUNG
   RUNG wire#powerrail
      Contact( "PLC_BIT".SIM )
      { S7_GenerateENO := "TRUE" } Move(in := "PLC_DATA".SI_WAG, out1 => "C#7_RD_RUN".WE_AG1)
      { S7_GenerateENO := "TRUE" } Move(in := "PLC_DATA".SI_WFD, out1 => "C#7_RD_RUN".WE_FD1)
      { S7_GenerateENO := "TRUE" } Move(in := "PLC_DATA".SI_WAP, out1 => "C#7_RD_RUN".WE_AP1)
      { S7_GenerateENO := "TRUE" } Move(in := "PLC_DATA".SI_WSB, out1 => "C#7_RD_RUN".WE_SB1)
   END_RUNG
   RUNG wire#powerrail
      I_Contact( "PLC_BIT".SIM )
      { S7_GenerateENO := "TRUE" } Move(in := "PLC_DATA".RE_WAG, out1 => "C#7_RD_RUN".WE_AG1)
      { S7_GenerateENO := "TRUE" } Move(in := "PLC_DATA".RE_WFD, out1 => "C#7_RD_RUN".WE_FD1)
      { S7_GenerateENO := "TRUE" } Move(in := "PLC_DATA".RE_WAP, out1 => "C#7_RD_RUN".WE_AP1)
      { S7_GenerateENO := "TRUE" } Move(in := "PLC_DATA".RE_WSB, out1 => "C#7_RD_RUN".WE_SB1)
   END_RUNG
   RUNG wire#powerrail
      Contact( "C#2_WB".F3_NN_STOP )
      wire#w2
      R_Coil( "PLC_BIT".RUN )
      R_Coil( "NAP LIEU" )
      R_Coil( "TH_NAP_WFD" )
      R_Coil( "TH_NAP_WSB" )
      R_Coil( "TH_NAP_WAP" )
      R_Coil( "TH_NAP_WAG" )
   END_RUNG
   RUNG wire#powerrail
      { S7_Templates := "SrcType := Real" } EQ_Contact(in1 := "C#7_RD_RUN".SMC_MIXER, in2 := "C#7_RD_RUN".SMT)
   END_RUNG wire#w2
   RUNG wire#w2
      { S7_GenerateENO := "TRUE" } Move(in := 0.0, out1 => "C#7_RD_RUN".SMC_AG1, out2 => "C#7_RD_RUN".SMX_AG1, out3 => "C#7_RD_RUN".SMC_AP1, out4 => "C#7_RD_RUN".SMX_AP1, out5 => "C#7_RD_RUN".SMC_FD1, out6 => "C#7_RD_RUN".SMX_FD1, out7 => "C#7_RD_RUN".SMC_SB1, out8 => "C#7_RD_RUN".SMX_SB1, out9 => "C#7_RD_RUN".SMC_MIXER, out10 => "C#7_RD_RUN".SMX_MIXER)
      { S7_GenerateENO := "TRUE" } Move(in := 0.0, out1 => "PLC_DATA".SMC_SILO_AG1, out2 => "PLC_DATA".SMC_SILO_AG2, out3 => "PLC_DATA".SMC_SILO_AG3, out4 => "PLC_DATA".SMC_SILO_AG4, out5 => "PLC_DATA".SMC_SILO_AG5, out6 => "PLC_DATA".SMC_SILO_FD1, out7 => "PLC_DATA".SMC_SILO_AP1, out8 => "PLC_DATA".SMC_SILO_SB1)
   END_RUNG
   RUNG wire#powerrail
      Move(in := "C#4_WD_WEIGHT".SO_ME_TRON, out1 => "C#7_RD_RUN".SMT)
   END_RUNG
   // the same network as SCL:
   // ENO of a box is taken as its EN; it also drops when the box reports an error
   IF "C#2_WB".F1_NN_RUN THEN "PLC_BIT".RUN := TRUE; END_IF;
   "P_RUN" := "C#2_WB".F1_NN_RUN;
   "PLC_BIT".SIM := "C#2_WB".F4_SW_SIM;
   "C#1_RB".RUNNING := "PLC_BIT".RUN;
   "C#1_RB".SIMULATION := "PLC_BIT".SIM;
   "PLC_BIT".AUT := "C#2_WB"."SW_MAN/AUTO";
   "PLC_BIT".MAN := NOT "C#2_WB"."SW_MAN/AUTO";
   IF "PLC_BIT".SIM THEN
       "C#7_RD_RUN".WE_AG1 := "PLC_DATA".SI_WAG;
       "C#7_RD_RUN".WE_FD1 := "PLC_DATA".SI_WFD;
       "C#7_RD_RUN".WE_AP1 := "PLC_DATA".SI_WAP;
       "C#7_RD_RUN".WE_SB1 := "PLC_DATA".SI_WSB;
   END_IF;
   IF NOT "PLC_BIT".SIM THEN
       "C#7_RD_RUN".WE_AG1 := "PLC_DATA".RE_WAG;
       "C#7_RD_RUN".WE_FD1 := "PLC_DATA".RE_WFD;
       "C#7_RD_RUN".WE_AP1 := "PLC_DATA".RE_WAP;
       "C#7_RD_RUN".WE_SB1 := "PLC_DATA".RE_WSB;
   END_IF;
   IF "C#2_WB".F3_NN_STOP OR ("C#7_RD_RUN".SMC_MIXER = "C#7_RD_RUN".SMT) THEN
       "PLC_BIT".RUN := FALSE;
       "NAP LIEU" := FALSE;
       "TH_NAP_WFD" := FALSE;
       "TH_NAP_WSB" := FALSE;
       "TH_NAP_WAP" := FALSE;
       "TH_NAP_WAG" := FALSE;
   END_IF;
   #_w1 := "C#2_WB".F3_NN_STOP OR ("C#7_RD_RUN".SMC_MIXER = "C#7_RD_RUN".SMT);
   IF #_w1 THEN
       "C#7_RD_RUN".SMC_AG1 := 0.0;
       "C#7_RD_RUN".SMX_AG1 := 0.0;
       "C#7_RD_RUN".SMC_AP1 := 0.0;
       "C#7_RD_RUN".SMX_AP1 := 0.0;
       "C#7_RD_RUN".SMC_FD1 := 0.0;
       "C#7_RD_RUN".SMX_FD1 := 0.0;
       "C#7_RD_RUN".SMC_SB1 := 0.0;
       "C#7_RD_RUN".SMX_SB1 := 0.0;
       "C#7_RD_RUN".SMC_MIXER := 0.0;
       "C#7_RD_RUN".SMX_MIXER := 0.0;
       "PLC_DATA".SMC_SILO_AG1 := 0.0;
       "PLC_DATA".SMC_SILO_AG2 := 0.0;
       "PLC_DATA".SMC_SILO_AG3 := 0.0;
       "PLC_DATA".SMC_SILO_AG4 := 0.0;
       "PLC_DATA".SMC_SILO_AG5 := 0.0;
       "PLC_DATA".SMC_SILO_FD1 := 0.0;
       "PLC_DATA".SMC_SILO_AP1 := 0.0;
       "PLC_DATA".SMC_SILO_SB1 := 0.0;
   END_IF;
   "C#7_RD_RUN".SMT := "C#4_WD_WEIGHT".SO_ME_TRON;
END_REGION

REGION Network 7: DATA SIMULATION
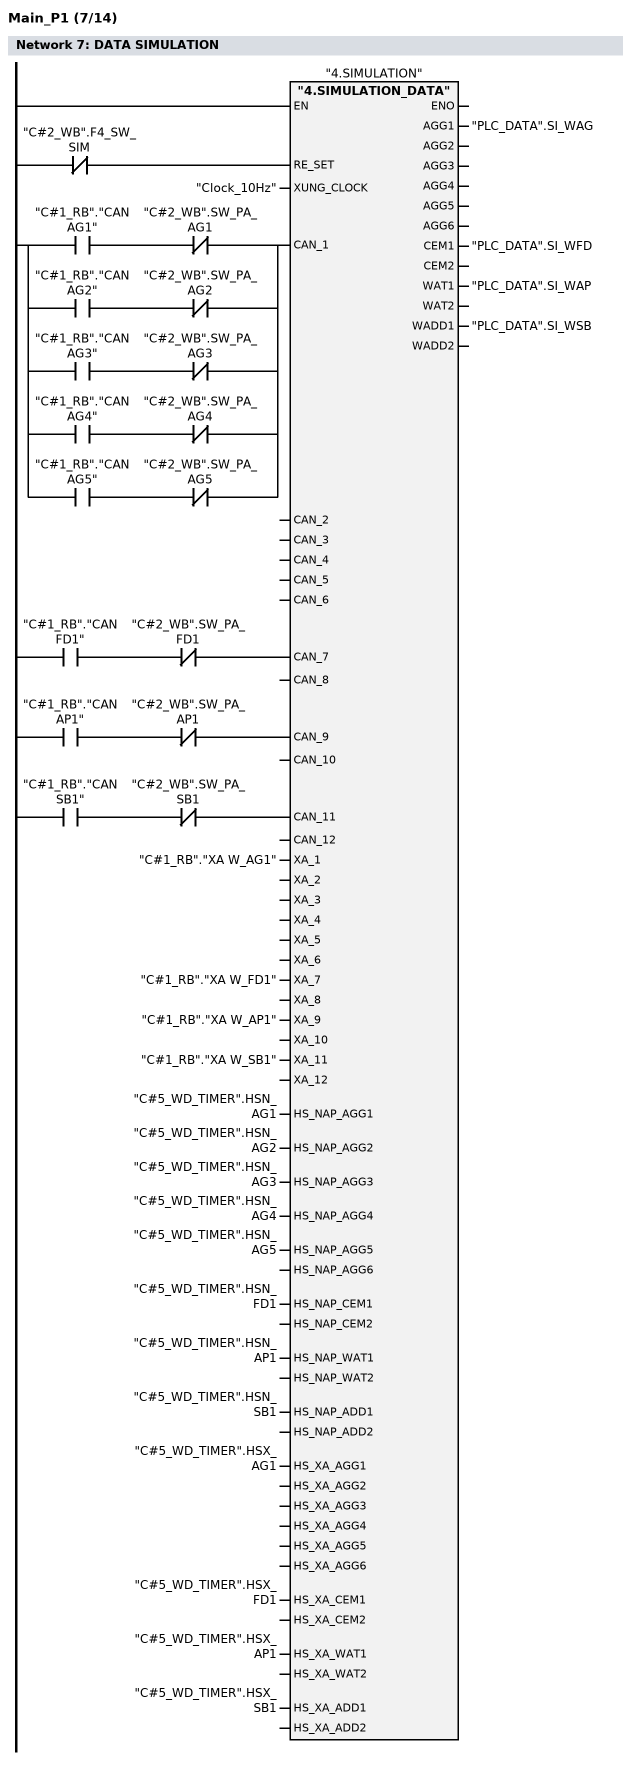
   RUNG wire#powerrail
      "4.SIMULATION"(RE_SET := wire#w1, CAN_1 := wire#w2, CAN_7 := wire#w3, CAN_9 := wire#w4, CAN_11 := wire#w5, XUNG_CLOCK := "Clock_10Hz", CAN_2 :=, CAN_3 :=, CAN_4 :=, CAN_5 :=, CAN_6 :=, CAN_8 :=, CAN_10 :=, CAN_12 :=, XA_1 := "C#1_RB"."XA W_AG1", XA_2 :=, XA_3 :=, XA_4 :=, XA_5 :=, XA_6 :=, XA_7 := "C#1_RB"."XA W_FD1", XA_8 :=, XA_9 := "C#1_RB"."XA W_AP1", XA_10 :=, XA_11 := "C#1_RB"."XA W_SB1", XA_12 :=, HS_NAP_AGG1 := "C#5_WD_TIMER".HSN_AG1, HS_NAP_AGG2 := "C#5_WD_TIMER".HSN_AG2, HS_NAP_AGG3 := "C#5_WD_TIMER".HSN_AG3, HS_NAP_AGG4 := "C#5_WD_TIMER".HSN_AG4, HS_NAP_AGG5 := "C#5_WD_TIMER".HSN_AG5, HS_NAP_AGG6 :=, HS_NAP_CEM1 := "C#5_WD_TIMER".HSN_FD1, HS_NAP_CEM2 :=, HS_NAP_WAT1 := "C#5_WD_TIMER".HSN_AP1, HS_NAP_WAT2 :=, HS_NAP_ADD1 := "C#5_WD_TIMER".HSN_SB1, HS_NAP_ADD2 :=, HS_XA_AGG1 := "C#5_WD_TIMER".HSX_AG1, HS_XA_AGG2 :=, HS_XA_AGG3 :=, HS_XA_AGG4 :=, HS_XA_AGG5 :=, HS_XA_AGG6 :=, HS_XA_CEM1 := "C#5_WD_TIMER".HSX_FD1, HS_XA_CEM2 :=, HS_XA_WAT1 := "C#5_WD_TIMER".HSX_AP1, HS_XA_WAT2 :=, HS_XA_ADD1 := "C#5_WD_TIMER".HSX_SB1, HS_XA_ADD2 :=, AGG1 => "PLC_DATA".SI_WAG, AGG2 =>, AGG3 =>, AGG4 =>, AGG5 =>, AGG6 =>, CEM1 => "PLC_DATA".SI_WFD, CEM2 =>, WAT1 => "PLC_DATA".SI_WAP, WAT2 =>, WADD1 => "PLC_DATA".SI_WSB, WADD2 =>)
   END_RUNG
   RUNG wire#powerrail
      I_Contact( "C#2_WB".F4_SW_SIM )
   END_RUNG wire#w1
   RUNG wire#powerrail
      Contact( "C#1_RB"."CAN AG1" )
      I_Contact( "C#2_WB".SW_PA_AG1 )
   END_RUNG wire#w2
   RUNG wire#powerrail
      Contact( "C#1_RB"."CAN AG2" )
      I_Contact( "C#2_WB".SW_PA_AG2 )
   END_RUNG wire#w2
   RUNG wire#powerrail
      Contact( "C#1_RB"."CAN AG3" )
      I_Contact( "C#2_WB".SW_PA_AG3 )
   END_RUNG wire#w2
   RUNG wire#powerrail
      Contact( "C#1_RB"."CAN AG4" )
      I_Contact( "C#2_WB".SW_PA_AG4 )
   END_RUNG wire#w2
   RUNG wire#powerrail
      Contact( "C#1_RB"."CAN AG5" )
      I_Contact( "C#2_WB".SW_PA_AG5 )
   END_RUNG wire#w2
   RUNG wire#powerrail
      Contact( "C#1_RB"."CAN FD1" )
      I_Contact( "C#2_WB".SW_PA_FD1 )
   END_RUNG wire#w3
   RUNG wire#powerrail
      Contact( "C#1_RB"."CAN AP1" )
      I_Contact( "C#2_WB".SW_PA_AP1 )
   END_RUNG wire#w4
   RUNG wire#powerrail
      Contact( "C#1_RB"."CAN SB1" )
      I_Contact( "C#2_WB".SW_PA_SB1 )
   END_RUNG wire#w5
   // the same network as SCL:
   "4.SIMULATION"(RE_SET := NOT "C#2_WB".F4_SW_SIM,   // "4.SIMULATION_DATA"
                  XUNG_CLOCK := "Clock_10Hz",
                  CAN_1 := ("C#1_RB"."CAN AG1" AND NOT "C#2_WB".SW_PA_AG1) OR ("C#1_RB"."CAN AG2" AND NOT "C#2_WB".SW_PA_AG2) OR ("C#1_RB"."CAN AG3" AND NOT "C#2_WB".SW_PA_AG3) OR ("C#1_RB"."CAN AG4" AND NOT "C#2_WB".SW_PA_AG4) OR ("C#1_RB"."CAN AG5" AND NOT "C#2_WB".SW_PA_AG5),
                  CAN_7 := "C#1_RB"."CAN FD1" AND NOT "C#2_WB".SW_PA_FD1,
                  CAN_9 := "C#1_RB"."CAN AP1" AND NOT "C#2_WB".SW_PA_AP1,
                  CAN_11 := "C#1_RB"."CAN SB1" AND NOT "C#2_WB".SW_PA_SB1,
                  XA_1 := "C#1_RB"."XA W_AG1",
                  XA_7 := "C#1_RB"."XA W_FD1",
                  XA_9 := "C#1_RB"."XA W_AP1",
                  XA_11 := "C#1_RB"."XA W_SB1",
                  HS_NAP_AGG1 := "C#5_WD_TIMER".HSN_AG1,
                  HS_NAP_AGG2 := "C#5_WD_TIMER".HSN_AG2,
                  HS_NAP_AGG3 := "C#5_WD_TIMER".HSN_AG3,
                  HS_NAP_AGG4 := "C#5_WD_TIMER".HSN_AG4,
                  HS_NAP_AGG5 := "C#5_WD_TIMER".HSN_AG5,
                  HS_NAP_CEM1 := "C#5_WD_TIMER".HSN_FD1,
                  HS_NAP_WAT1 := "C#5_WD_TIMER".HSN_AP1,
                  HS_NAP_ADD1 := "C#5_WD_TIMER".HSN_SB1,
                  HS_XA_AGG1 := "C#5_WD_TIMER".HSX_AG1,
                  HS_XA_CEM1 := "C#5_WD_TIMER".HSX_FD1,
                  HS_XA_WAT1 := "C#5_WD_TIMER".HSX_AP1,
                  HS_XA_ADD1 := "C#5_WD_TIMER".HSX_SB1,
                  AGG1 => "PLC_DATA".SI_WAG,
                  CEM1 => "PLC_DATA".SI_WFD,
                  WAT1 => "PLC_DATA".SI_WAP,
                  WADD1 => "PLC_DATA".SI_WSB);
END_REGION

REGION Network 8: XỬ LÍ CÂN CỐT LIỆU
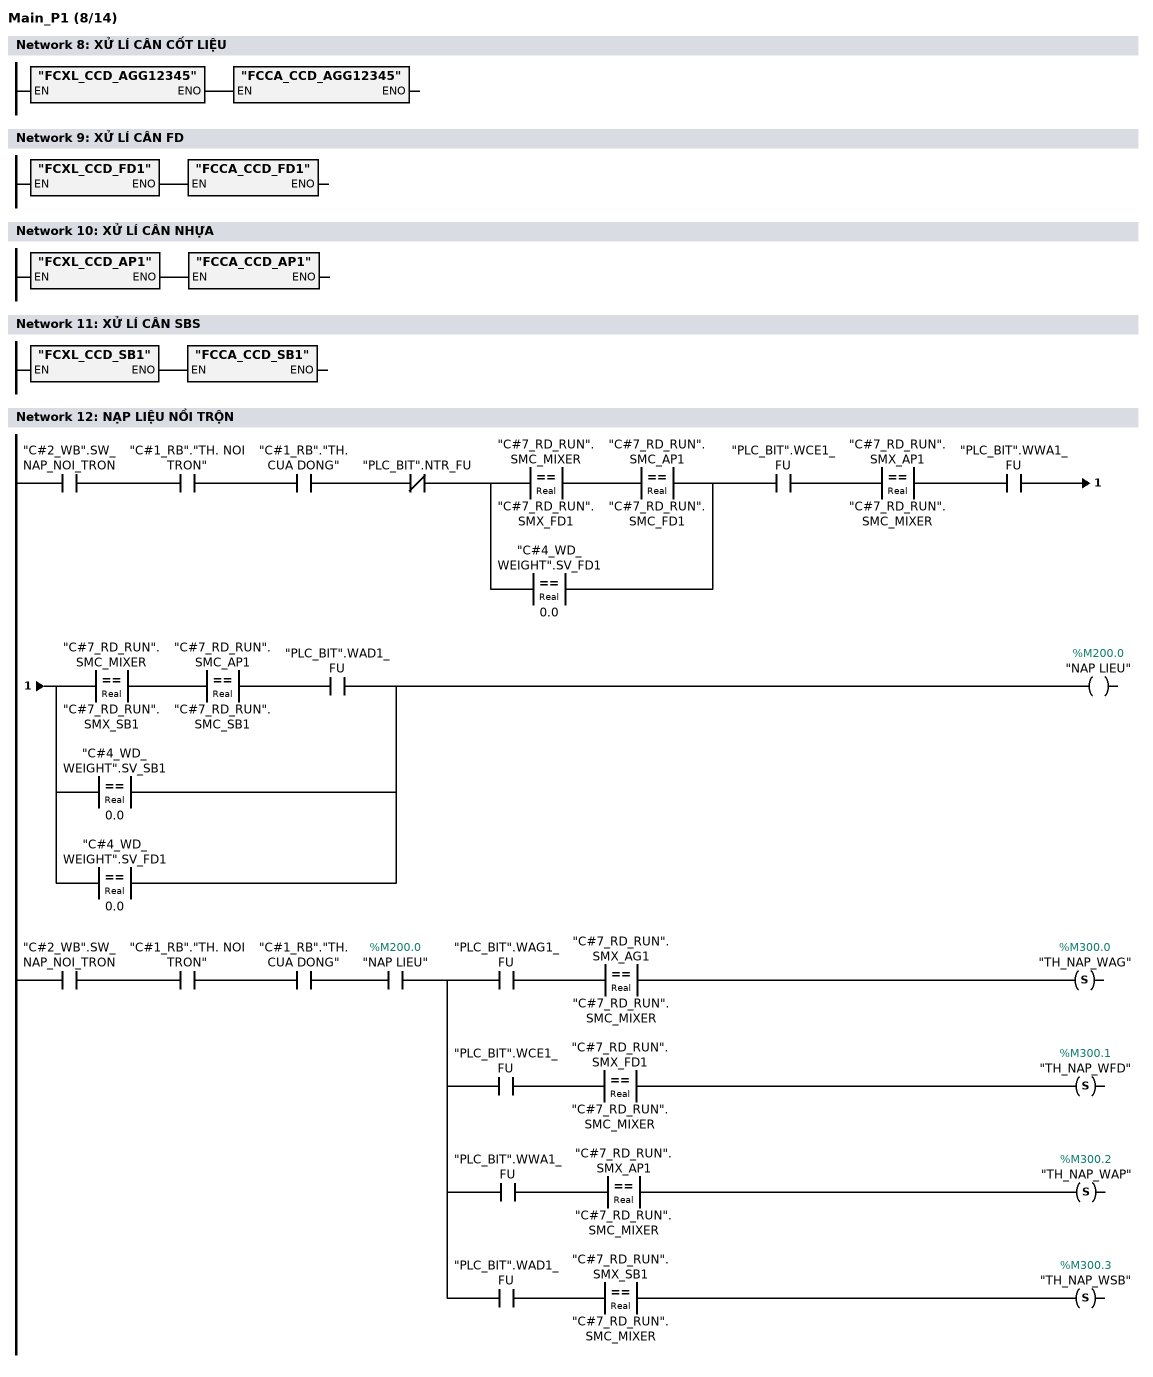
   RUNG wire#powerrail
      "FCXL_CCD_AGG12345"()
      "FCCA_CCD_AGG12345"()
   END_RUNG
   // the same network as SCL:
   "FCXL_CCD_AGG12345"(ENO => #_w1);
   IF #_w1 THEN "FCCA_CCD_AGG12345"(); END_IF;
END_REGION

REGION Network 9: XỬ LÍ CÂN FD
   RUNG wire#powerrail
      "FCXL_CCD_FD1"()
      "FCCA_CCD_FD1"()
   END_RUNG
   // the same network as SCL:
   "FCXL_CCD_FD1"(ENO => #_w1);
   IF #_w1 THEN "FCCA_CCD_FD1"(); END_IF;
END_REGION

REGION Network 10: XỬ LÍ CÂN NHỰA
   RUNG wire#powerrail
      "FCXL_CCD_AP1"()
      "FCCA_CCD_AP1"()
   END_RUNG
   // the same network as SCL:
   "FCXL_CCD_AP1"(ENO => #_w1);
   IF #_w1 THEN "FCCA_CCD_AP1"(); END_IF;
END_REGION

REGION Network 11: XỬ LÍ CÂN SBS
   RUNG wire#powerrail
      "FCXL_CCD_SB1"()
      "FCCA_CCD_SB1"()
   END_RUNG
   // the same network as SCL:
   "FCXL_CCD_SB1"(ENO => #_w1);
   IF #_w1 THEN "FCCA_CCD_SB1"(); END_IF;
END_REGION

REGION Network 12: NẠP LIỆU NỒI TRỘN
   RUNG wire#powerrail
      Contact( "C#2_WB".SW_NAP_NOI_TRON )
      Contact( "C#1_RB"."TH. NOI TRON" )
      Contact( "C#1_RB"."TH. CUA DONG" )
      I_Contact( "PLC_BIT".NTR_FU )
      wire#w1
      { S7_Templates := "SrcType := Real" } EQ_Contact(in1 := "C#7_RD_RUN".SMC_MIXER, in2 := "C#7_RD_RUN".SMX_FD1)
      { S7_Templates := "SrcType := Real" } EQ_Contact(in1 := "C#7_RD_RUN".SMC_AP1, in2 := "C#7_RD_RUN".SMC_FD1)
      wire#w2
      Contact( "PLC_BIT".WCE1_FU )
      { S7_Templates := "SrcType := Real" } EQ_Contact(in1 := "C#7_RD_RUN".SMX_AP1, in2 := "C#7_RD_RUN".SMC_MIXER)
      Contact( "PLC_BIT".WWA1_FU )
      wire#w3
      { S7_Templates := "SrcType := Real" } EQ_Contact(in1 := "C#7_RD_RUN".SMC_MIXER, in2 := "C#7_RD_RUN".SMX_SB1)
      { S7_Templates := "SrcType := Real" } EQ_Contact(in1 := "C#7_RD_RUN".SMC_AP1, in2 := "C#7_RD_RUN".SMC_SB1)
      Contact( "PLC_BIT".WAD1_FU )
      wire#w4
      Coil( "NAP LIEU" )
   END_RUNG
   RUNG wire#w1
      { S7_Templates := "SrcType := Real" } EQ_Contact(in1 := "C#4_WD_WEIGHT".SV_FD1, in2 := 0.0)
   END_RUNG wire#w2
   RUNG wire#w3
      { S7_Templates := "SrcType := Real" } EQ_Contact(in1 := "C#4_WD_WEIGHT".SV_SB1, in2 := 0.0)
   END_RUNG wire#w4
   RUNG wire#w3
      { S7_Templates := "SrcType := Real" } EQ_Contact(in1 := "C#4_WD_WEIGHT".SV_FD1, in2 := 0.0)
   END_RUNG wire#w4
   RUNG wire#powerrail
      Contact( "C#2_WB".SW_NAP_NOI_TRON )
      Contact( "C#1_RB"."TH. NOI TRON" )
      Contact( "C#1_RB"."TH. CUA DONG" )
      Contact( "NAP LIEU" )
      wire#w5
      Contact( "PLC_BIT".WAG1_FU )
      { S7_Templates := "SrcType := Real" } EQ_Contact(in1 := "C#7_RD_RUN".SMX_AG1, in2 := "C#7_RD_RUN".SMC_MIXER)
      S_Coil( "TH_NAP_WAG" )
   END_RUNG
   RUNG wire#w5
      Contact( "PLC_BIT".WCE1_FU )
      { S7_Templates := "SrcType := Real" } EQ_Contact(in1 := "C#7_RD_RUN".SMX_FD1, in2 := "C#7_RD_RUN".SMC_MIXER)
      S_Coil( "TH_NAP_WFD" )
   END_RUNG
   RUNG wire#w5
      Contact( "PLC_BIT".WWA1_FU )
      { S7_Templates := "SrcType := Real" } EQ_Contact(in1 := "C#7_RD_RUN".SMX_AP1, in2 := "C#7_RD_RUN".SMC_MIXER)
      S_Coil( "TH_NAP_WAP" )
   END_RUNG
   RUNG wire#w5
      Contact( "PLC_BIT".WAD1_FU )
      { S7_Templates := "SrcType := Real" } EQ_Contact(in1 := "C#7_RD_RUN".SMX_SB1, in2 := "C#7_RD_RUN".SMC_MIXER)
      S_Coil( "TH_NAP_WSB" )
   END_RUNG
   // the same network as SCL:
   "NAP LIEU" := "C#2_WB".SW_NAP_NOI_TRON AND "C#1_RB"."TH. NOI TRON" AND "C#1_RB"."TH. CUA DONG" AND NOT "PLC_BIT".NTR_FU AND ((("C#7_RD_RUN".SMC_MIXER = "C#7_RD_RUN".SMX_FD1) AND ("C#7_RD_RUN".SMC_AP1 = "C#7_RD_RUN".SMC_FD1)) OR ("C#4_WD_WEIGHT".SV_FD1 = 0.0)) AND "PLC_BIT".WCE1_FU AND ("C#7_RD_RUN".SMX_AP1 = "C#7_RD_RUN".SMC_MIXER) AND "PLC_BIT".WWA1_FU AND ((("C#7_RD_RUN".SMC_MIXER = "C#7_RD_RUN".SMX_SB1) AND ("C#7_RD_RUN".SMC_AP1 = "C#7_RD_RUN".SMC_SB1) AND "PLC_BIT".WAD1_FU) OR ("C#4_WD_WEIGHT".SV_SB1 = 0.0) OR ("C#4_WD_WEIGHT".SV_FD1 = 0.0));
   #_w1 := "C#2_WB".SW_NAP_NOI_TRON AND "C#1_RB"."TH. NOI TRON" AND "C#1_RB"."TH. CUA DONG" AND "NAP LIEU";
   IF #_w1 AND "PLC_BIT".WAG1_FU AND ("C#7_RD_RUN".SMX_AG1 = "C#7_RD_RUN".SMC_MIXER) THEN
       "TH_NAP_WAG" := TRUE;
   END_IF;
   IF #_w1 AND "PLC_BIT".WCE1_FU AND ("C#7_RD_RUN".SMX_FD1 = "C#7_RD_RUN".SMC_MIXER) THEN
       "TH_NAP_WFD" := TRUE;
   END_IF;
   IF #_w1 AND "PLC_BIT".WWA1_FU AND ("C#7_RD_RUN".SMX_AP1 = "C#7_RD_RUN".SMC_MIXER) THEN
       "TH_NAP_WAP" := TRUE;
   END_IF;
   IF #_w1 AND "PLC_BIT".WAD1_FU AND ("C#7_RD_RUN".SMX_SB1 = "C#7_RD_RUN".SMC_MIXER) THEN
       "TH_NAP_WSB" := TRUE;
   END_IF;
END_REGION

REGION Network 13: XỬ LÍ NỒI TRỘN
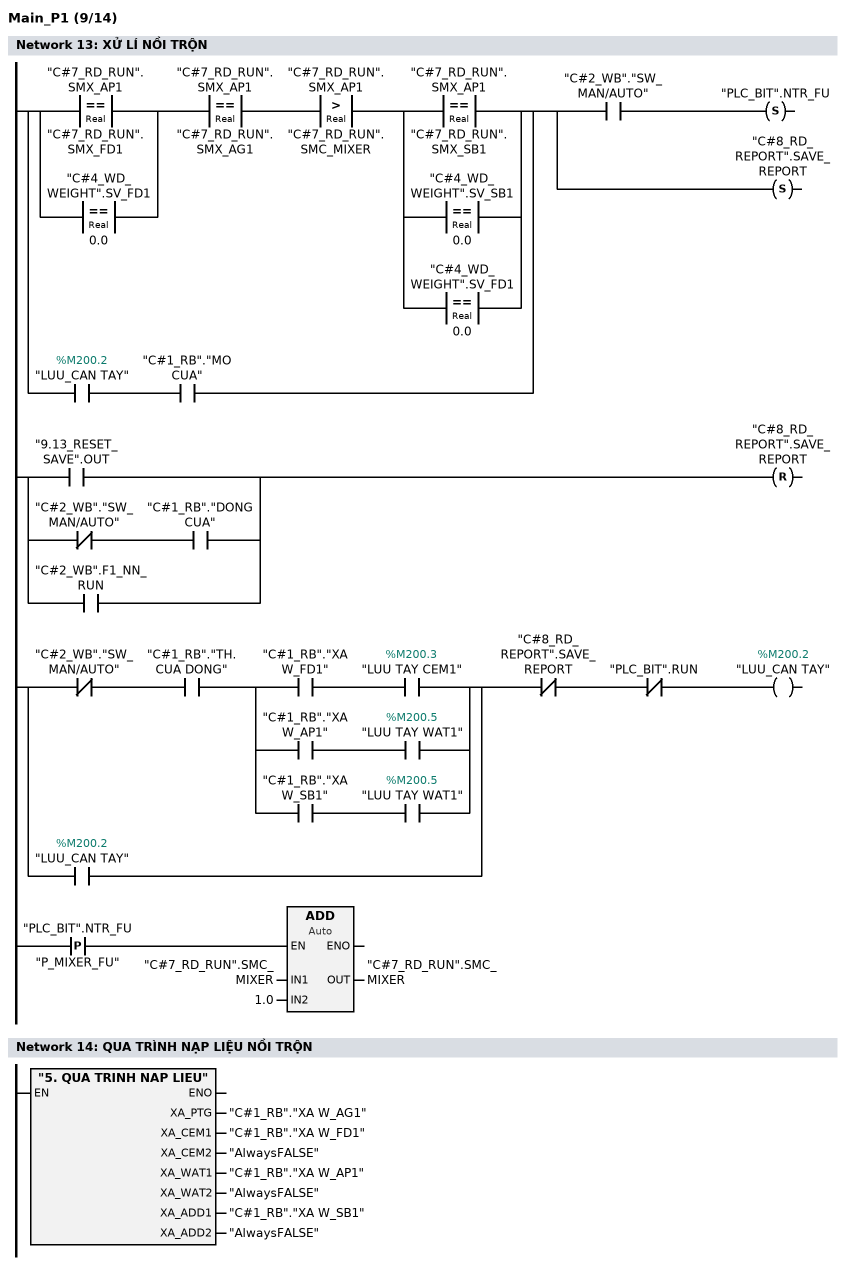
   RUNG wire#powerrail
      { S7_Templates := "SrcType := Real" } EQ_Contact(in1 := "C#7_RD_RUN".SMX_AP1, in2 := "C#7_RD_RUN".SMX_FD1)
      wire#w1
      { S7_Templates := "SrcType := Real" } EQ_Contact(in1 := "C#7_RD_RUN".SMX_AP1, in2 := "C#7_RD_RUN".SMX_AG1)
      { S7_Templates := "SrcType := Real" } GT_Contact(in1 := "C#7_RD_RUN".SMX_AP1, in2 := "C#7_RD_RUN".SMC_MIXER)
      wire#w2
      { S7_Templates := "SrcType := Real" } EQ_Contact(in1 := "C#7_RD_RUN".SMX_AP1, in2 := "C#7_RD_RUN".SMX_SB1)
      wire#w3
      Contact( "C#2_WB"."SW_MAN/AUTO" )
      S_Coil( "PLC_BIT".NTR_FU )
   END_RUNG
   RUNG wire#powerrail
      { S7_Templates := "SrcType := Real" } EQ_Contact(in1 := "C#4_WD_WEIGHT".SV_FD1, in2 := 0.0)
   END_RUNG wire#w1
   RUNG wire#w2
      { S7_Templates := "SrcType := Real" } EQ_Contact(in1 := "C#4_WD_WEIGHT".SV_SB1, in2 := 0.0)
   END_RUNG wire#w3
   RUNG wire#w2
      { S7_Templates := "SrcType := Real" } EQ_Contact(in1 := "C#4_WD_WEIGHT".SV_FD1, in2 := 0.0)
   END_RUNG wire#w3
   RUNG wire#powerrail
      Contact( "LUU_CAN TAY" )
      Contact( "C#1_RB"."MO CUA" )
   END_RUNG wire#w3
   RUNG wire#w3
      S_Coil( "C#8_RD_REPORT".SAVE_REPORT )
   END_RUNG
   RUNG wire#powerrail
      Contact( "9.13_RESET_SAVE".OUT )
      wire#w4
      R_Coil( "C#8_RD_REPORT".SAVE_REPORT )
   END_RUNG
   RUNG wire#powerrail
      I_Contact( "C#2_WB"."SW_MAN/AUTO" )
      Contact( "C#1_RB"."DONG CUA" )
   END_RUNG wire#w4
   RUNG wire#powerrail
      Contact( "C#2_WB".F1_NN_RUN )
   END_RUNG wire#w4
   RUNG wire#powerrail
      I_Contact( "C#2_WB"."SW_MAN/AUTO" )
      Contact( "C#1_RB"."TH. CUA DONG" )
      wire#w5
      Contact( "C#1_RB"."XA W_FD1" )
      Contact( "LUU TAY CEM1" )
      wire#w6
      I_Contact( "C#8_RD_REPORT".SAVE_REPORT )
      I_Contact( "PLC_BIT".RUN )
      Coil( "LUU_CAN TAY" )
   END_RUNG
   RUNG wire#w5
      Contact( "C#1_RB"."XA W_AP1" )
      Contact( "LUU TAY WAT1" )
   END_RUNG wire#w6
   RUNG wire#w5
      Contact( "C#1_RB"."XA W_SB1" )
      Contact( "LUU TAY WAT1" )
   END_RUNG wire#w6
   RUNG wire#powerrail
      Contact( "LUU_CAN TAY" )
   END_RUNG wire#w6
   RUNG wire#powerrail
      P_Contact(operand := "PLC_BIT".NTR_FU, bit := "P_MIXER_FU")
      Add(in1 := "C#7_RD_RUN".SMC_MIXER, in2 := 1.0, out => "C#7_RD_RUN".SMC_MIXER)
   END_RUNG
   // the same network as SCL:
   #_w1 := ((("C#7_RD_RUN".SMX_AP1 = "C#7_RD_RUN".SMX_FD1) OR ("C#4_WD_WEIGHT".SV_FD1 = 0.0)) AND ("C#7_RD_RUN".SMX_AP1 = "C#7_RD_RUN".SMX_AG1) AND ("C#7_RD_RUN".SMX_AP1 > "C#7_RD_RUN".SMC_MIXER) AND (("C#7_RD_RUN".SMX_AP1 = "C#7_RD_RUN".SMX_SB1) OR ("C#4_WD_WEIGHT".SV_SB1 = 0.0) OR ("C#4_WD_WEIGHT".SV_FD1 = 0.0))) OR ("LUU_CAN TAY" AND "C#1_RB"."MO CUA");
   IF #_w1 AND "C#2_WB"."SW_MAN/AUTO" THEN "PLC_BIT".NTR_FU := TRUE; END_IF;
   IF #_w1 THEN "C#8_RD_REPORT".SAVE_REPORT := TRUE; END_IF;
   IF "9.13_RESET_SAVE".OUT OR (NOT "C#2_WB"."SW_MAN/AUTO" AND "C#1_RB"."DONG CUA") OR "C#2_WB".F1_NN_RUN THEN
       "C#8_RD_REPORT".SAVE_REPORT := FALSE;
   END_IF;
   "LUU_CAN TAY" := ((NOT "C#2_WB"."SW_MAN/AUTO" AND "C#1_RB"."TH. CUA DONG" AND (("C#1_RB"."XA W_FD1" AND "LUU TAY CEM1") OR ("C#1_RB"."XA W_AP1" AND "LUU TAY WAT1") OR ("C#1_RB"."XA W_SB1" AND "LUU TAY WAT1"))) OR "LUU_CAN TAY") AND NOT "C#8_RD_REPORT".SAVE_REPORT AND NOT "PLC_BIT".RUN;
   #_w2 := "PLC_BIT".NTR_FU AND NOT "P_MIXER_FU";   // rising edge of "PLC_BIT".NTR_FU
   "P_MIXER_FU" := "PLC_BIT".NTR_FU;
   IF #_w2 THEN "C#7_RD_RUN".SMC_MIXER := "C#7_RD_RUN".SMC_MIXER + 1.0; END_IF;
END_REGION

REGION Network 14: QUA TRÌNH NẠP LIỆU NỒI TRỘN
   RUNG wire#powerrail
      "5. QUA TRINH NAP LIEU"(XA_PTG => "C#1_RB"."XA W_AG1", XA_CEM1 => "C#1_RB"."XA W_FD1", XA_CEM2 => "AlwaysFALSE", XA_WAT1 => "C#1_RB"."XA W_AP1", XA_WAT2 => "AlwaysFALSE", XA_ADD1 => "C#1_RB"."XA W_SB1", XA_ADD2 => "AlwaysFALSE")
   END_RUNG
   // the same network as SCL:
   "5. QUA TRINH NAP LIEU"(XA_PTG => "C#1_RB"."XA W_AG1",
                           XA_CEM1 => "C#1_RB"."XA W_FD1",
                           XA_CEM2 => "AlwaysFALSE",
                           XA_WAT1 => "C#1_RB"."XA W_AP1",
                           XA_WAT2 => "AlwaysFALSE",
                           XA_ADD1 => "C#1_RB"."XA W_SB1",
                           XA_ADD2 => "AlwaysFALSE");
END_REGION

